// TIA Portal V20 export
FUNCTION_BLOCK "EventsPFE"   // FB74, LAD
AUTHOR : ERsystem_FA2_DH. Kim
// stored: IsIECCheckEnabled true, MemoryReserve 100, Namespace Unit1.Em6, SetENOAutomatically false
   VAR
      data : Array[1..100] of LReal;
   END_VAR
BEGIN

REGION Network 1: Call PFE Events
   // Add the required PFE Events
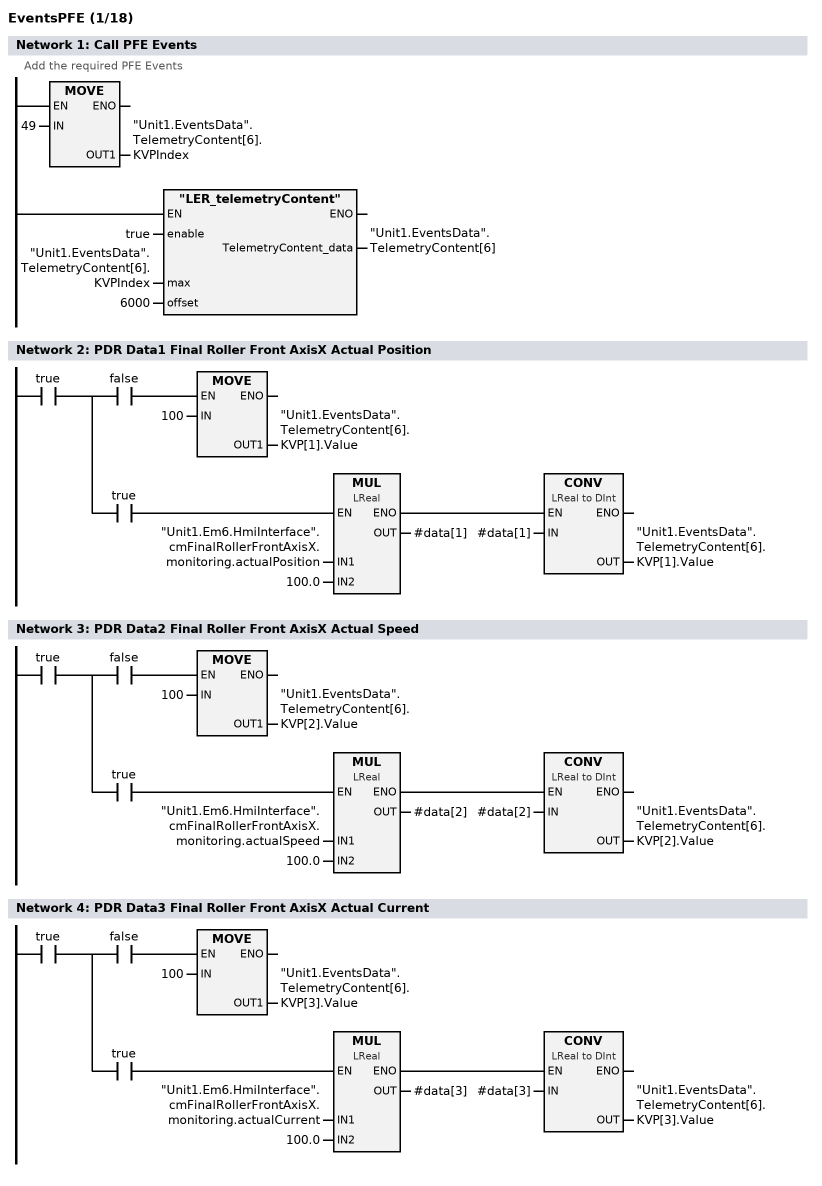
   RUNG wire#powerrail
      Move(in := 49, out1 => "Unit1.EventsData".TelemetryContent[6].KVPIndex)
   END_RUNG
   RUNG wire#powerrail
      "LER_telemetryContent"(enable := true, max := "Unit1.EventsData".TelemetryContent[6].KVPIndex, offset := 6000, TelemetryContent_data => "Unit1.EventsData".TelemetryContent[6])
   END_RUNG
   // the same network as SCL:
   "Unit1.EventsData".TelemetryContent[6].KVPIndex := 49;
   "LER_telemetryContent"(enable := true,
                          max := "Unit1.EventsData".TelemetryContent[6].KVPIndex,
                          offset := 6000,
                          TelemetryContent_data => "Unit1.EventsData".TelemetryContent[6]);
END_REGION

REGION Network 2: PDR Data1 Final Roller Front AxisX Actual Position
   RUNG wire#powerrail
      Contact( true )
      wire#w1
      Contact( false )
      Move(in := 100, out1 => "Unit1.EventsData".TelemetryContent[6].KVP[1].Value)
   END_RUNG
   RUNG wire#w1
      Contact( true )
      { S7_Templates := "SrcType := LReal" } Mul(in1 := "Unit1.Em6.HmiInterface".cmFinalRollerFrontAxisX.monitoring.actualPosition, in2 := 100.0, out => #data[1])
      { S7_Templates := "[SrcType := LReal, DestType := DInt]" } Convert(in := #data[1], out => "Unit1.EventsData".TelemetryContent[6].KVP[1].Value)
   END_RUNG
   // the same network as SCL:
   IF true AND false THEN "Unit1.EventsData".TelemetryContent[6].KVP[1].Value := 100; END_IF;
   IF true AND true THEN
       #data[1] := "Unit1.Em6.HmiInterface".cmFinalRollerFrontAxisX.monitoring.actualPosition * 100.0;
       "Unit1.EventsData".TelemetryContent[6].KVP[1].Value := LREAL_TO_DINT(#data[1]);
   END_IF;
END_REGION

REGION Network 3: PDR Data2 Final Roller Front AxisX Actual Speed
   RUNG wire#powerrail
      Contact( true )
      wire#w1
      Contact( false )
      Move(in := 100, out1 => "Unit1.EventsData".TelemetryContent[6].KVP[2].Value)
   END_RUNG
   RUNG wire#w1
      Contact( true )
      { S7_Templates := "SrcType := LReal" } Mul(in1 := "Unit1.Em6.HmiInterface".cmFinalRollerFrontAxisX.monitoring.actualSpeed, in2 := 100.0, out => #data[2])
      { S7_Templates := "[SrcType := LReal, DestType := DInt]" } Convert(in := #data[2], out => "Unit1.EventsData".TelemetryContent[6].KVP[2].Value)
   END_RUNG
   // the same network as SCL:
   IF true AND false THEN "Unit1.EventsData".TelemetryContent[6].KVP[2].Value := 100; END_IF;
   IF true AND true THEN
       #data[2] := "Unit1.Em6.HmiInterface".cmFinalRollerFrontAxisX.monitoring.actualSpeed * 100.0;
       "Unit1.EventsData".TelemetryContent[6].KVP[2].Value := LREAL_TO_DINT(#data[2]);
   END_IF;
END_REGION

REGION Network 4: PDR Data3 Final Roller Front AxisX Actual Current
   RUNG wire#powerrail
      Contact( true )
      wire#w1
      Contact( false )
      Move(in := 100, out1 => "Unit1.EventsData".TelemetryContent[6].KVP[3].Value)
   END_RUNG
   RUNG wire#w1
      Contact( true )
      { S7_Templates := "SrcType := LReal" } Mul(in1 := "Unit1.Em6.HmiInterface".cmFinalRollerFrontAxisX.monitoring.actualCurrent, in2 := 100.0, out => #data[3])
      { S7_Templates := "[SrcType := LReal, DestType := DInt]" } Convert(in := #data[3], out => "Unit1.EventsData".TelemetryContent[6].KVP[3].Value)
   END_RUNG
   // the same network as SCL:
   IF true AND false THEN "Unit1.EventsData".TelemetryContent[6].KVP[3].Value := 100; END_IF;
   IF true AND true THEN
       #data[3] := "Unit1.Em6.HmiInterface".cmFinalRollerFrontAxisX.monitoring.actualCurrent * 100.0;
       "Unit1.EventsData".TelemetryContent[6].KVP[3].Value := LREAL_TO_DINT(#data[3]);
   END_IF;
END_REGION

REGION Network 5: PDR Data4 Final Roller Front AxisX Actual Torque
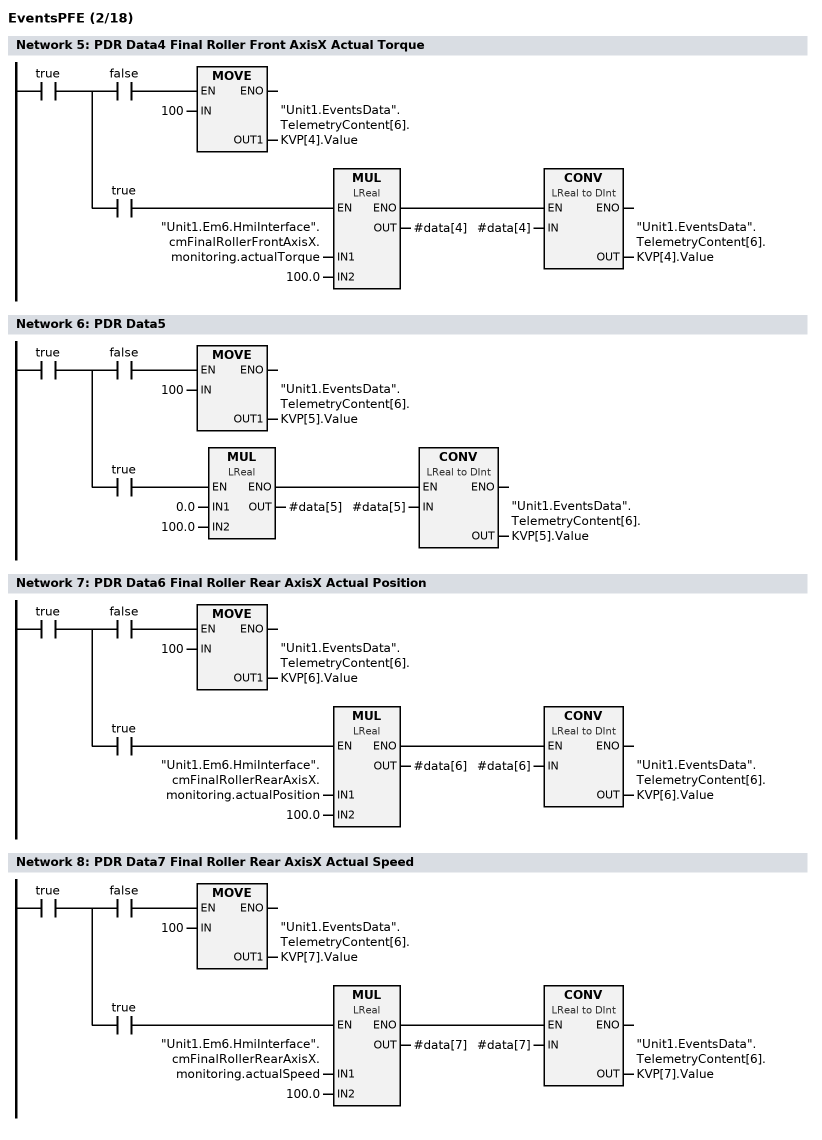
   RUNG wire#powerrail
      Contact( true )
      wire#w1
      Contact( false )
      Move(in := 100, out1 => "Unit1.EventsData".TelemetryContent[6].KVP[4].Value)
   END_RUNG
   RUNG wire#w1
      Contact( true )
      { S7_Templates := "SrcType := LReal" } Mul(in1 := "Unit1.Em6.HmiInterface".cmFinalRollerFrontAxisX.monitoring.actualTorque, in2 := 100.0, out => #data[4])
      { S7_Templates := "[SrcType := LReal, DestType := DInt]" } Convert(in := #data[4], out => "Unit1.EventsData".TelemetryContent[6].KVP[4].Value)
   END_RUNG
   // the same network as SCL:
   IF true AND false THEN "Unit1.EventsData".TelemetryContent[6].KVP[4].Value := 100; END_IF;
   IF true AND true THEN
       #data[4] := "Unit1.Em6.HmiInterface".cmFinalRollerFrontAxisX.monitoring.actualTorque * 100.0;
       "Unit1.EventsData".TelemetryContent[6].KVP[4].Value := LREAL_TO_DINT(#data[4]);
   END_IF;
END_REGION

REGION Network 6: PDR Data5
   RUNG wire#powerrail
      Contact( true )
      wire#w1
      Contact( false )
      Move(in := 100, out1 => "Unit1.EventsData".TelemetryContent[6].KVP[5].Value)
   END_RUNG
   RUNG wire#w1
      Contact( true )
      { S7_Templates := "SrcType := LReal" } Mul(in1 := 0.0, in2 := 100.0, out => #data[5])
      { S7_Templates := "[SrcType := LReal, DestType := DInt]" } Convert(in := #data[5], out => "Unit1.EventsData".TelemetryContent[6].KVP[5].Value)
   END_RUNG
   // the same network as SCL:
   IF true AND false THEN "Unit1.EventsData".TelemetryContent[6].KVP[5].Value := 100; END_IF;
   IF true AND true THEN
       #data[5] := 0.0 * 100.0;
       "Unit1.EventsData".TelemetryContent[6].KVP[5].Value := LREAL_TO_DINT(#data[5]);
   END_IF;
END_REGION

REGION Network 7: PDR Data6 Final Roller Rear AxisX Actual Position
   RUNG wire#powerrail
      Contact( true )
      wire#w1
      Contact( false )
      Move(in := 100, out1 => "Unit1.EventsData".TelemetryContent[6].KVP[6].Value)
   END_RUNG
   RUNG wire#w1
      Contact( true )
      { S7_Templates := "SrcType := LReal" } Mul(in1 := "Unit1.Em6.HmiInterface".cmFinalRollerRearAxisX.monitoring.actualPosition, in2 := 100.0, out => #data[6])
      { S7_Templates := "[SrcType := LReal, DestType := DInt]" } Convert(in := #data[6], out => "Unit1.EventsData".TelemetryContent[6].KVP[6].Value)
   END_RUNG
   // the same network as SCL:
   IF true AND false THEN "Unit1.EventsData".TelemetryContent[6].KVP[6].Value := 100; END_IF;
   IF true AND true THEN
       #data[6] := "Unit1.Em6.HmiInterface".cmFinalRollerRearAxisX.monitoring.actualPosition * 100.0;
       "Unit1.EventsData".TelemetryContent[6].KVP[6].Value := LREAL_TO_DINT(#data[6]);
   END_IF;
END_REGION

REGION Network 8: PDR Data7 Final Roller Rear AxisX Actual Speed
   RUNG wire#powerrail
      Contact( true )
      wire#w1
      Contact( false )
      Move(in := 100, out1 => "Unit1.EventsData".TelemetryContent[6].KVP[7].Value)
   END_RUNG
   RUNG wire#w1
      Contact( true )
      { S7_Templates := "SrcType := LReal" } Mul(in1 := "Unit1.Em6.HmiInterface".cmFinalRollerRearAxisX.monitoring.actualSpeed, in2 := 100.0, out => #data[7])
      { S7_Templates := "[SrcType := LReal, DestType := DInt]" } Convert(in := #data[7], out => "Unit1.EventsData".TelemetryContent[6].KVP[7].Value)
   END_RUNG
   // the same network as SCL:
   IF true AND false THEN "Unit1.EventsData".TelemetryContent[6].KVP[7].Value := 100; END_IF;
   IF true AND true THEN
       #data[7] := "Unit1.Em6.HmiInterface".cmFinalRollerRearAxisX.monitoring.actualSpeed * 100.0;
       "Unit1.EventsData".TelemetryContent[6].KVP[7].Value := LREAL_TO_DINT(#data[7]);
   END_IF;
END_REGION

REGION Network 9: PDR Data8 Final Roller Rear AxisX Actual Current
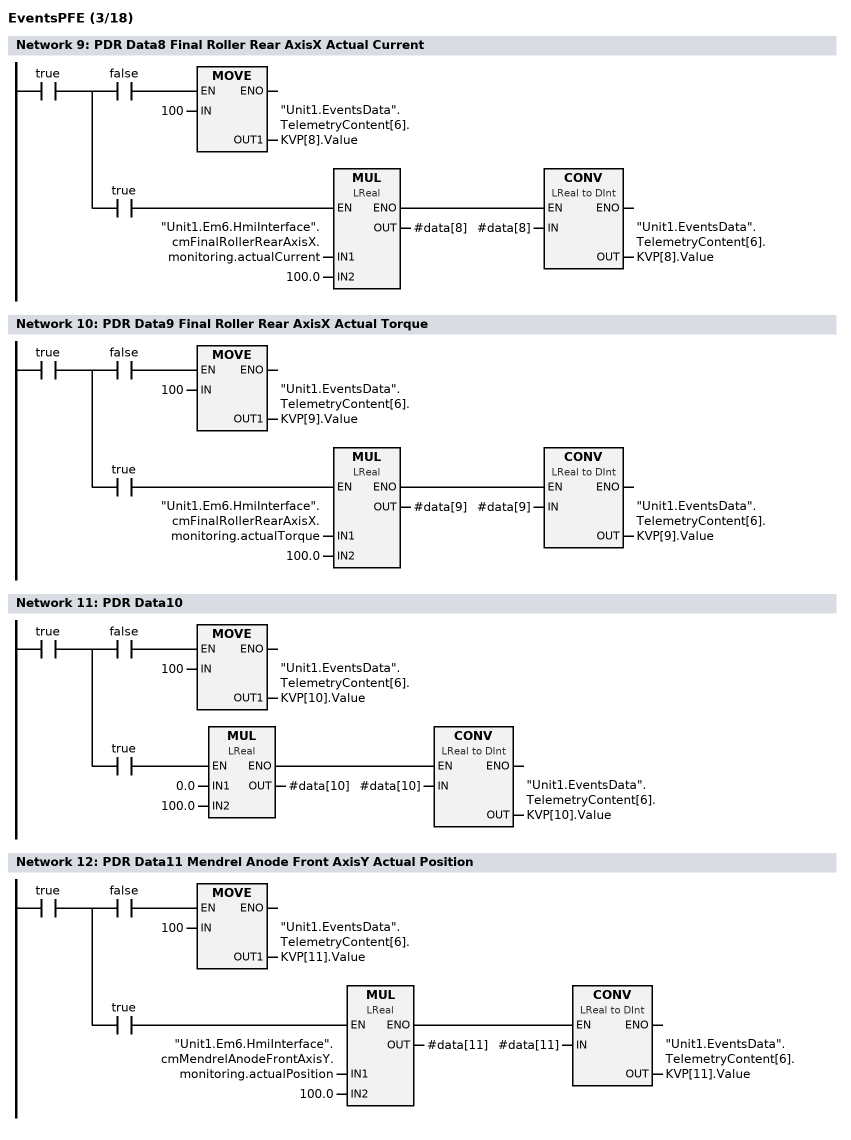
   RUNG wire#powerrail
      Contact( true )
      wire#w1
      Contact( false )
      Move(in := 100, out1 => "Unit1.EventsData".TelemetryContent[6].KVP[8].Value)
   END_RUNG
   RUNG wire#w1
      Contact( true )
      { S7_Templates := "SrcType := LReal" } Mul(in1 := "Unit1.Em6.HmiInterface".cmFinalRollerRearAxisX.monitoring.actualCurrent, in2 := 100.0, out => #data[8])
      { S7_Templates := "[SrcType := LReal, DestType := DInt]" } Convert(in := #data[8], out => "Unit1.EventsData".TelemetryContent[6].KVP[8].Value)
   END_RUNG
   // the same network as SCL:
   IF true AND false THEN "Unit1.EventsData".TelemetryContent[6].KVP[8].Value := 100; END_IF;
   IF true AND true THEN
       #data[8] := "Unit1.Em6.HmiInterface".cmFinalRollerRearAxisX.monitoring.actualCurrent * 100.0;
       "Unit1.EventsData".TelemetryContent[6].KVP[8].Value := LREAL_TO_DINT(#data[8]);
   END_IF;
END_REGION

REGION Network 10: PDR Data9 Final Roller Rear AxisX Actual Torque
   RUNG wire#powerrail
      Contact( true )
      wire#w1
      Contact( false )
      Move(in := 100, out1 => "Unit1.EventsData".TelemetryContent[6].KVP[9].Value)
   END_RUNG
   RUNG wire#w1
      Contact( true )
      { S7_Templates := "SrcType := LReal" } Mul(in1 := "Unit1.Em6.HmiInterface".cmFinalRollerRearAxisX.monitoring.actualTorque, in2 := 100.0, out => #data[9])
      { S7_Templates := "[SrcType := LReal, DestType := DInt]" } Convert(in := #data[9], out => "Unit1.EventsData".TelemetryContent[6].KVP[9].Value)
   END_RUNG
   // the same network as SCL:
   IF true AND false THEN "Unit1.EventsData".TelemetryContent[6].KVP[9].Value := 100; END_IF;
   IF true AND true THEN
       #data[9] := "Unit1.Em6.HmiInterface".cmFinalRollerRearAxisX.monitoring.actualTorque * 100.0;
       "Unit1.EventsData".TelemetryContent[6].KVP[9].Value := LREAL_TO_DINT(#data[9]);
   END_IF;
END_REGION

REGION Network 11: PDR Data10
   RUNG wire#powerrail
      Contact( true )
      wire#w1
      Contact( false )
      Move(in := 100, out1 => "Unit1.EventsData".TelemetryContent[6].KVP[10].Value)
   END_RUNG
   RUNG wire#w1
      Contact( true )
      { S7_Templates := "SrcType := LReal" } Mul(in1 := 0.0, in2 := 100.0, out => #data[10])
      { S7_Templates := "[SrcType := LReal, DestType := DInt]" } Convert(in := #data[10], out => "Unit1.EventsData".TelemetryContent[6].KVP[10].Value)
   END_RUNG
   // the same network as SCL:
   IF true AND false THEN "Unit1.EventsData".TelemetryContent[6].KVP[10].Value := 100; END_IF;
   IF true AND true THEN
       #data[10] := 0.0 * 100.0;
       "Unit1.EventsData".TelemetryContent[6].KVP[10].Value := LREAL_TO_DINT(#data[10]);
   END_IF;
END_REGION

REGION Network 12: PDR Data11 Mendrel Anode Front AxisY Actual Position
   RUNG wire#powerrail
      Contact( true )
      wire#w1
      Contact( false )
      Move(in := 100, out1 => "Unit1.EventsData".TelemetryContent[6].KVP[11].Value)
   END_RUNG
   RUNG wire#w1
      Contact( true )
      { S7_Templates := "SrcType := LReal" } Mul(in1 := "Unit1.Em6.HmiInterface".cmMendrelAnodeFrontAxisY.monitoring.actualPosition, in2 := 100.0, out => #data[11])
      { S7_Templates := "[SrcType := LReal, DestType := DInt]" } Convert(in := #data[11], out => "Unit1.EventsData".TelemetryContent[6].KVP[11].Value)
   END_RUNG
   // the same network as SCL:
   IF true AND false THEN "Unit1.EventsData".TelemetryContent[6].KVP[11].Value := 100; END_IF;
   IF true AND true THEN
       #data[11] := "Unit1.Em6.HmiInterface".cmMendrelAnodeFrontAxisY.monitoring.actualPosition * 100.0;
       "Unit1.EventsData".TelemetryContent[6].KVP[11].Value := LREAL_TO_DINT(#data[11]);
   END_IF;
END_REGION

REGION Network 13: PDR Data12 Mendrel Anode Front AxisY Actual Speed
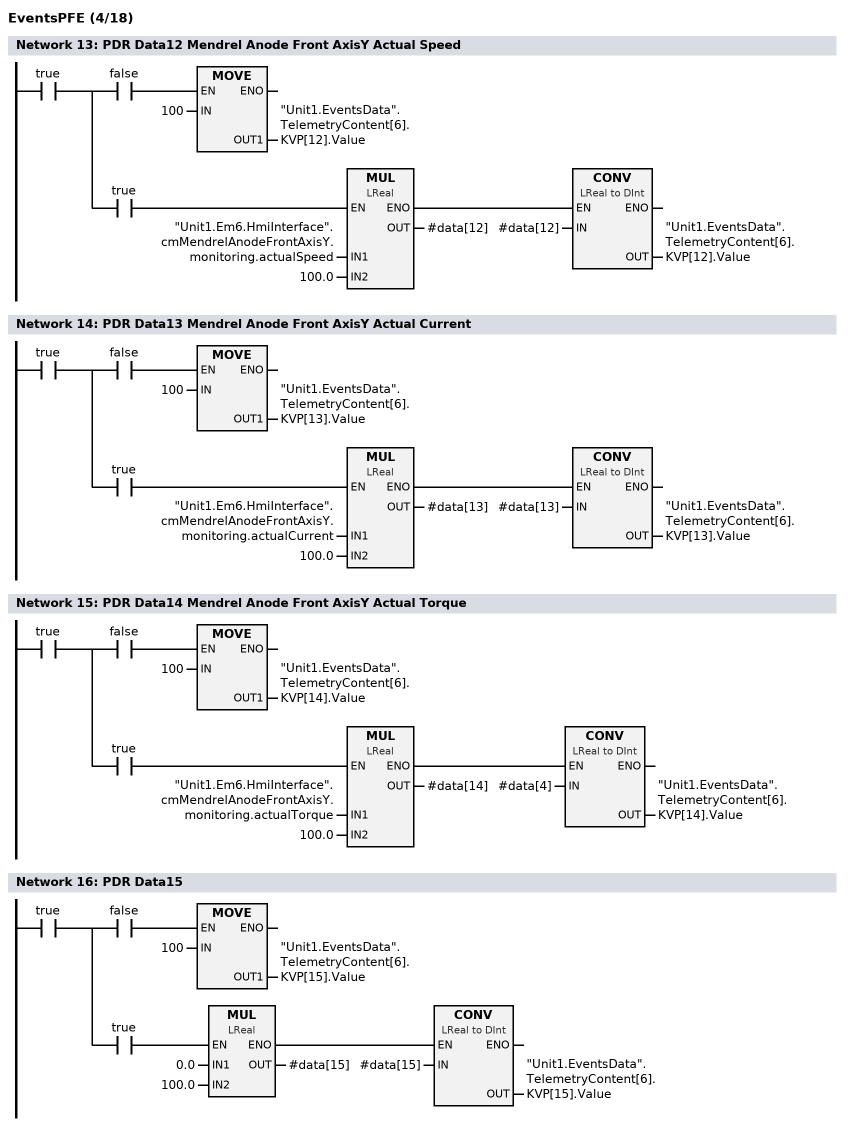
   RUNG wire#powerrail
      Contact( true )
      wire#w1
      Contact( false )
      Move(in := 100, out1 => "Unit1.EventsData".TelemetryContent[6].KVP[12].Value)
   END_RUNG
   RUNG wire#w1
      Contact( true )
      { S7_Templates := "SrcType := LReal" } Mul(in1 := "Unit1.Em6.HmiInterface".cmMendrelAnodeFrontAxisY.monitoring.actualSpeed, in2 := 100.0, out => #data[12])
      { S7_Templates := "[SrcType := LReal, DestType := DInt]" } Convert(in := #data[12], out => "Unit1.EventsData".TelemetryContent[6].KVP[12].Value)
   END_RUNG
   // the same network as SCL:
   IF true AND false THEN "Unit1.EventsData".TelemetryContent[6].KVP[12].Value := 100; END_IF;
   IF true AND true THEN
       #data[12] := "Unit1.Em6.HmiInterface".cmMendrelAnodeFrontAxisY.monitoring.actualSpeed * 100.0;
       "Unit1.EventsData".TelemetryContent[6].KVP[12].Value := LREAL_TO_DINT(#data[12]);
   END_IF;
END_REGION

REGION Network 14: PDR Data13 Mendrel Anode Front AxisY Actual Current
   RUNG wire#powerrail
      Contact( true )
      wire#w1
      Contact( false )
      Move(in := 100, out1 => "Unit1.EventsData".TelemetryContent[6].KVP[13].Value)
   END_RUNG
   RUNG wire#w1
      Contact( true )
      { S7_Templates := "SrcType := LReal" } Mul(in1 := "Unit1.Em6.HmiInterface".cmMendrelAnodeFrontAxisY.monitoring.actualCurrent, in2 := 100.0, out => #data[13])
      { S7_Templates := "[SrcType := LReal, DestType := DInt]" } Convert(in := #data[13], out => "Unit1.EventsData".TelemetryContent[6].KVP[13].Value)
   END_RUNG
   // the same network as SCL:
   IF true AND false THEN "Unit1.EventsData".TelemetryContent[6].KVP[13].Value := 100; END_IF;
   IF true AND true THEN
       #data[13] := "Unit1.Em6.HmiInterface".cmMendrelAnodeFrontAxisY.monitoring.actualCurrent * 100.0;
       "Unit1.EventsData".TelemetryContent[6].KVP[13].Value := LREAL_TO_DINT(#data[13]);
   END_IF;
END_REGION

REGION Network 15: PDR Data14 Mendrel Anode Front AxisY Actual Torque
   RUNG wire#powerrail
      Contact( true )
      wire#w1
      Contact( false )
      Move(in := 100, out1 => "Unit1.EventsData".TelemetryContent[6].KVP[14].Value)
   END_RUNG
   RUNG wire#w1
      Contact( true )
      { S7_Templates := "SrcType := LReal" } Mul(in1 := "Unit1.Em6.HmiInterface".cmMendrelAnodeFrontAxisY.monitoring.actualTorque, in2 := 100.0, out => #data[14])
      { S7_Templates := "[SrcType := LReal, DestType := DInt]" } Convert(in := #data[4], out => "Unit1.EventsData".TelemetryContent[6].KVP[14].Value)
   END_RUNG
   // the same network as SCL:
   IF true AND false THEN "Unit1.EventsData".TelemetryContent[6].KVP[14].Value := 100; END_IF;
   IF true AND true THEN
       #data[14] := "Unit1.Em6.HmiInterface".cmMendrelAnodeFrontAxisY.monitoring.actualTorque * 100.0;
       "Unit1.EventsData".TelemetryContent[6].KVP[14].Value := LREAL_TO_DINT(#data[4]);
   END_IF;
END_REGION

REGION Network 16: PDR Data15
   RUNG wire#powerrail
      Contact( true )
      wire#w1
      Contact( false )
      Move(in := 100, out1 => "Unit1.EventsData".TelemetryContent[6].KVP[15].Value)
   END_RUNG
   RUNG wire#w1
      Contact( true )
      { S7_Templates := "SrcType := LReal" } Mul(in1 := 0.0, in2 := 100.0, out => #data[15])
      { S7_Templates := "[SrcType := LReal, DestType := DInt]" } Convert(in := #data[15], out => "Unit1.EventsData".TelemetryContent[6].KVP[15].Value)
   END_RUNG
   // the same network as SCL:
   IF true AND false THEN "Unit1.EventsData".TelemetryContent[6].KVP[15].Value := 100; END_IF;
   IF true AND true THEN
       #data[15] := 0.0 * 100.0;
       "Unit1.EventsData".TelemetryContent[6].KVP[15].Value := LREAL_TO_DINT(#data[15]);
   END_IF;
END_REGION

REGION Network 17: PDR Data16 Mendrel Anode Front AxisZ Actual Position
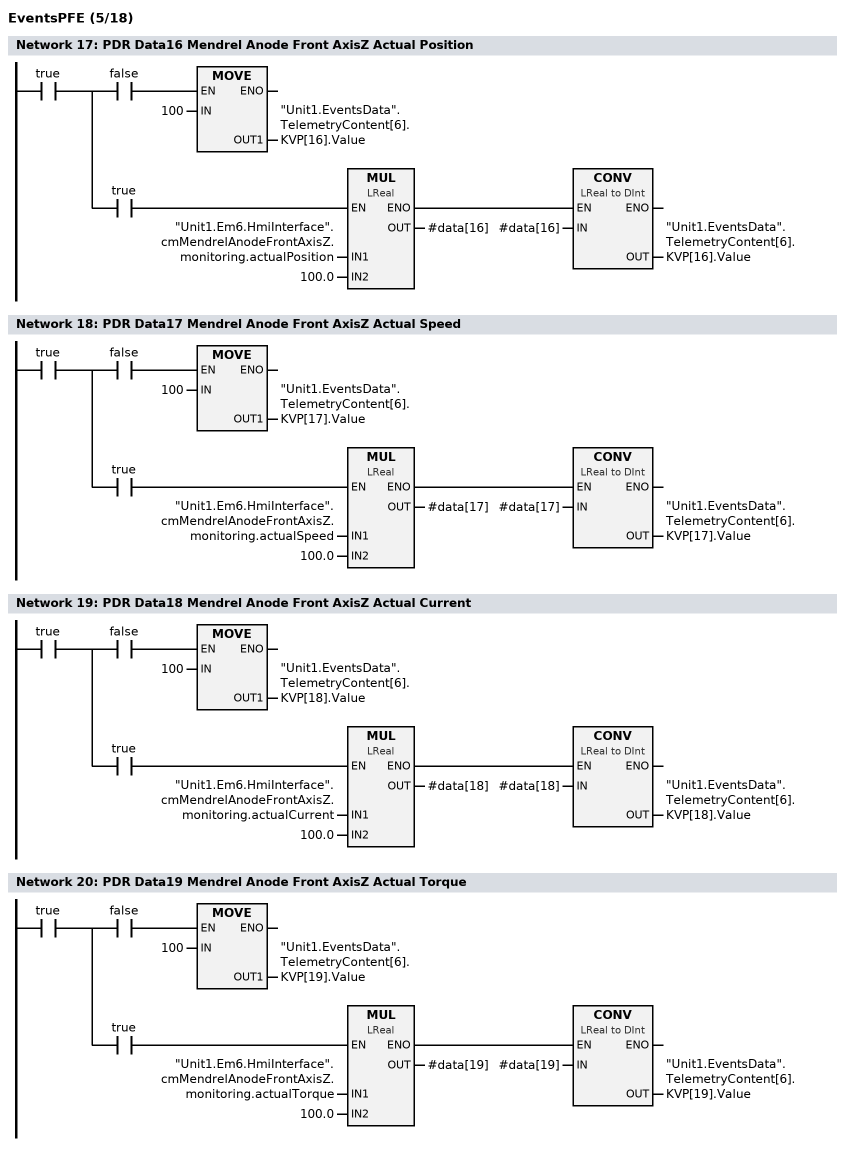
   RUNG wire#powerrail
      Contact( true )
      wire#w1
      Contact( false )
      Move(in := 100, out1 => "Unit1.EventsData".TelemetryContent[6].KVP[16].Value)
   END_RUNG
   RUNG wire#w1
      Contact( true )
      { S7_Templates := "SrcType := LReal" } Mul(in1 := "Unit1.Em6.HmiInterface".cmMendrelAnodeFrontAxisZ.monitoring.actualPosition, in2 := 100.0, out => #data[16])
      { S7_Templates := "[SrcType := LReal, DestType := DInt]" } Convert(in := #data[16], out => "Unit1.EventsData".TelemetryContent[6].KVP[16].Value)
   END_RUNG
   // the same network as SCL:
   IF true AND false THEN "Unit1.EventsData".TelemetryContent[6].KVP[16].Value := 100; END_IF;
   IF true AND true THEN
       #data[16] := "Unit1.Em6.HmiInterface".cmMendrelAnodeFrontAxisZ.monitoring.actualPosition * 100.0;
       "Unit1.EventsData".TelemetryContent[6].KVP[16].Value := LREAL_TO_DINT(#data[16]);
   END_IF;
END_REGION

REGION Network 18: PDR Data17 Mendrel Anode Front AxisZ Actual Speed
   RUNG wire#powerrail
      Contact( true )
      wire#w1
      Contact( false )
      Move(in := 100, out1 => "Unit1.EventsData".TelemetryContent[6].KVP[17].Value)
   END_RUNG
   RUNG wire#w1
      Contact( true )
      { S7_Templates := "SrcType := LReal" } Mul(in1 := "Unit1.Em6.HmiInterface".cmMendrelAnodeFrontAxisZ.monitoring.actualSpeed, in2 := 100.0, out => #data[17])
      { S7_Templates := "[SrcType := LReal, DestType := DInt]" } Convert(in := #data[17], out => "Unit1.EventsData".TelemetryContent[6].KVP[17].Value)
   END_RUNG
   // the same network as SCL:
   IF true AND false THEN "Unit1.EventsData".TelemetryContent[6].KVP[17].Value := 100; END_IF;
   IF true AND true THEN
       #data[17] := "Unit1.Em6.HmiInterface".cmMendrelAnodeFrontAxisZ.monitoring.actualSpeed * 100.0;
       "Unit1.EventsData".TelemetryContent[6].KVP[17].Value := LREAL_TO_DINT(#data[17]);
   END_IF;
END_REGION

REGION Network 19: PDR Data18 Mendrel Anode Front AxisZ Actual Current
   RUNG wire#powerrail
      Contact( true )
      wire#w1
      Contact( false )
      Move(in := 100, out1 => "Unit1.EventsData".TelemetryContent[6].KVP[18].Value)
   END_RUNG
   RUNG wire#w1
      Contact( true )
      { S7_Templates := "SrcType := LReal" } Mul(in1 := "Unit1.Em6.HmiInterface".cmMendrelAnodeFrontAxisZ.monitoring.actualCurrent, in2 := 100.0, out => #data[18])
      { S7_Templates := "[SrcType := LReal, DestType := DInt]" } Convert(in := #data[18], out => "Unit1.EventsData".TelemetryContent[6].KVP[18].Value)
   END_RUNG
   // the same network as SCL:
   IF true AND false THEN "Unit1.EventsData".TelemetryContent[6].KVP[18].Value := 100; END_IF;
   IF true AND true THEN
       #data[18] := "Unit1.Em6.HmiInterface".cmMendrelAnodeFrontAxisZ.monitoring.actualCurrent * 100.0;
       "Unit1.EventsData".TelemetryContent[6].KVP[18].Value := LREAL_TO_DINT(#data[18]);
   END_IF;
END_REGION

REGION Network 20: PDR Data19 Mendrel Anode Front AxisZ Actual Torque
   RUNG wire#powerrail
      Contact( true )
      wire#w1
      Contact( false )
      Move(in := 100, out1 => "Unit1.EventsData".TelemetryContent[6].KVP[19].Value)
   END_RUNG
   RUNG wire#w1
      Contact( true )
      { S7_Templates := "SrcType := LReal" } Mul(in1 := "Unit1.Em6.HmiInterface".cmMendrelAnodeFrontAxisZ.monitoring.actualTorque, in2 := 100.0, out => #data[19])
      { S7_Templates := "[SrcType := LReal, DestType := DInt]" } Convert(in := #data[19], out => "Unit1.EventsData".TelemetryContent[6].KVP[19].Value)
   END_RUNG
   // the same network as SCL:
   IF true AND false THEN "Unit1.EventsData".TelemetryContent[6].KVP[19].Value := 100; END_IF;
   IF true AND true THEN
       #data[19] := "Unit1.Em6.HmiInterface".cmMendrelAnodeFrontAxisZ.monitoring.actualTorque * 100.0;
       "Unit1.EventsData".TelemetryContent[6].KVP[19].Value := LREAL_TO_DINT(#data[19]);
   END_IF;
END_REGION

REGION Network 21: PDR Data20
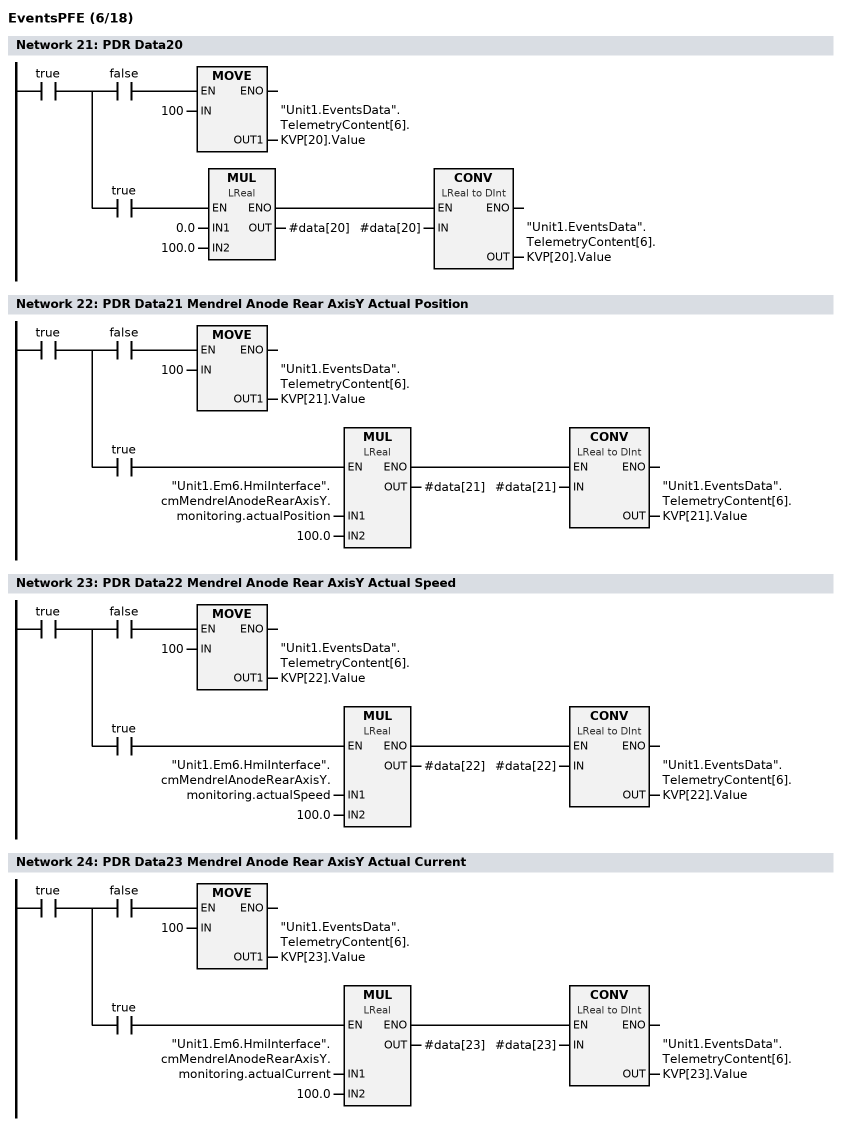
   RUNG wire#powerrail
      Contact( true )
      wire#w1
      Contact( false )
      Move(in := 100, out1 => "Unit1.EventsData".TelemetryContent[6].KVP[20].Value)
   END_RUNG
   RUNG wire#w1
      Contact( true )
      { S7_Templates := "SrcType := LReal" } Mul(in1 := 0.0, in2 := 100.0, out => #data[20])
      { S7_Templates := "[SrcType := LReal, DestType := DInt]" } Convert(in := #data[20], out => "Unit1.EventsData".TelemetryContent[6].KVP[20].Value)
   END_RUNG
   // the same network as SCL:
   IF true AND false THEN "Unit1.EventsData".TelemetryContent[6].KVP[20].Value := 100; END_IF;
   IF true AND true THEN
       #data[20] := 0.0 * 100.0;
       "Unit1.EventsData".TelemetryContent[6].KVP[20].Value := LREAL_TO_DINT(#data[20]);
   END_IF;
END_REGION

REGION Network 22: PDR Data21 Mendrel Anode Rear AxisY Actual Position
   RUNG wire#powerrail
      Contact( true )
      wire#w1
      Contact( false )
      Move(in := 100, out1 => "Unit1.EventsData".TelemetryContent[6].KVP[21].Value)
   END_RUNG
   RUNG wire#w1
      Contact( true )
      { S7_Templates := "SrcType := LReal" } Mul(in1 := "Unit1.Em6.HmiInterface".cmMendrelAnodeRearAxisY.monitoring.actualPosition, in2 := 100.0, out => #data[21])
      { S7_Templates := "[SrcType := LReal, DestType := DInt]" } Convert(in := #data[21], out => "Unit1.EventsData".TelemetryContent[6].KVP[21].Value)
   END_RUNG
   // the same network as SCL:
   IF true AND false THEN "Unit1.EventsData".TelemetryContent[6].KVP[21].Value := 100; END_IF;
   IF true AND true THEN
       #data[21] := "Unit1.Em6.HmiInterface".cmMendrelAnodeRearAxisY.monitoring.actualPosition * 100.0;
       "Unit1.EventsData".TelemetryContent[6].KVP[21].Value := LREAL_TO_DINT(#data[21]);
   END_IF;
END_REGION

REGION Network 23: PDR Data22 Mendrel Anode Rear AxisY Actual Speed
   RUNG wire#powerrail
      Contact( true )
      wire#w1
      Contact( false )
      Move(in := 100, out1 => "Unit1.EventsData".TelemetryContent[6].KVP[22].Value)
   END_RUNG
   RUNG wire#w1
      Contact( true )
      { S7_Templates := "SrcType := LReal" } Mul(in1 := "Unit1.Em6.HmiInterface".cmMendrelAnodeRearAxisY.monitoring.actualSpeed, in2 := 100.0, out => #data[22])
      { S7_Templates := "[SrcType := LReal, DestType := DInt]" } Convert(in := #data[22], out => "Unit1.EventsData".TelemetryContent[6].KVP[22].Value)
   END_RUNG
   // the same network as SCL:
   IF true AND false THEN "Unit1.EventsData".TelemetryContent[6].KVP[22].Value := 100; END_IF;
   IF true AND true THEN
       #data[22] := "Unit1.Em6.HmiInterface".cmMendrelAnodeRearAxisY.monitoring.actualSpeed * 100.0;
       "Unit1.EventsData".TelemetryContent[6].KVP[22].Value := LREAL_TO_DINT(#data[22]);
   END_IF;
END_REGION

REGION Network 24: PDR Data23 Mendrel Anode Rear AxisY Actual Current
   RUNG wire#powerrail
      Contact( true )
      wire#w1
      Contact( false )
      Move(in := 100, out1 => "Unit1.EventsData".TelemetryContent[6].KVP[23].Value)
   END_RUNG
   RUNG wire#w1
      Contact( true )
      { S7_Templates := "SrcType := LReal" } Mul(in1 := "Unit1.Em6.HmiInterface".cmMendrelAnodeRearAxisY.monitoring.actualCurrent, in2 := 100.0, out => #data[23])
      { S7_Templates := "[SrcType := LReal, DestType := DInt]" } Convert(in := #data[23], out => "Unit1.EventsData".TelemetryContent[6].KVP[23].Value)
   END_RUNG
   // the same network as SCL:
   IF true AND false THEN "Unit1.EventsData".TelemetryContent[6].KVP[23].Value := 100; END_IF;
   IF true AND true THEN
       #data[23] := "Unit1.Em6.HmiInterface".cmMendrelAnodeRearAxisY.monitoring.actualCurrent * 100.0;
       "Unit1.EventsData".TelemetryContent[6].KVP[23].Value := LREAL_TO_DINT(#data[23]);
   END_IF;
END_REGION

REGION Network 25: PDR Data24 Mendrel Anode Rear AxisY Actual Torque
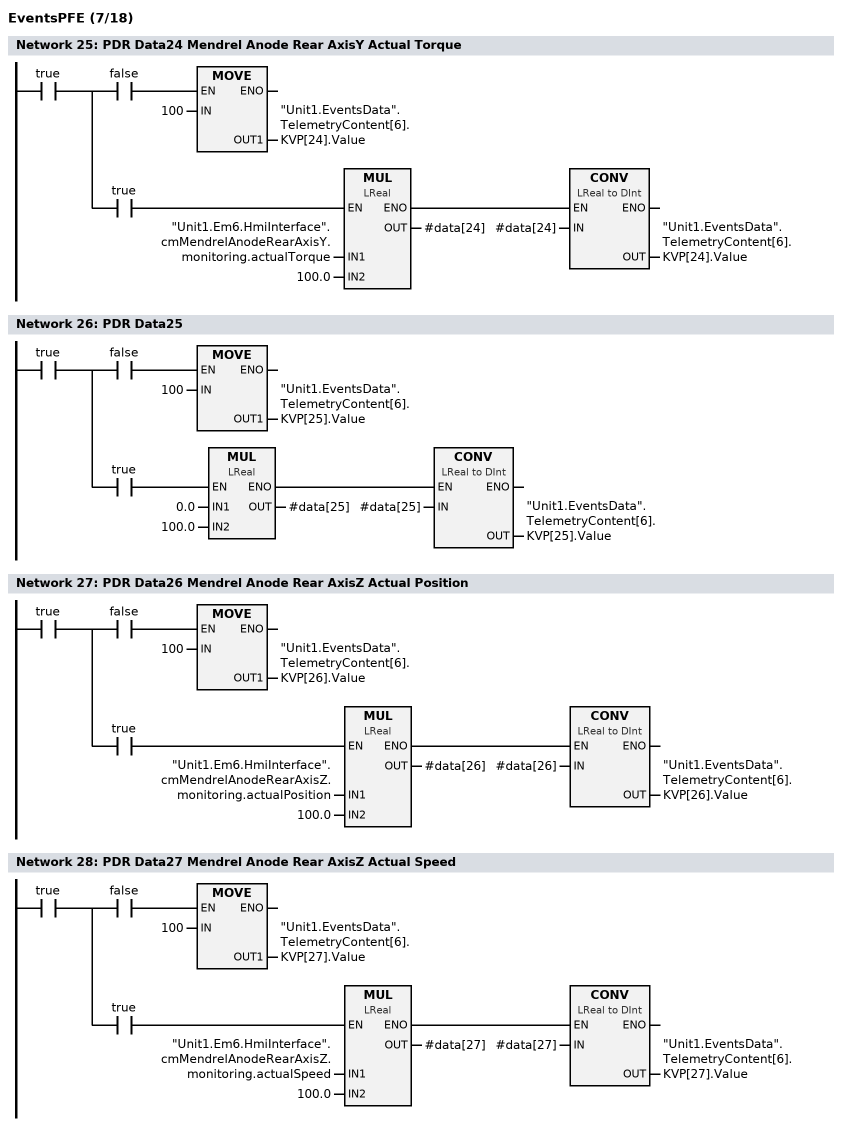
   RUNG wire#powerrail
      Contact( true )
      wire#w1
      Contact( false )
      Move(in := 100, out1 => "Unit1.EventsData".TelemetryContent[6].KVP[24].Value)
   END_RUNG
   RUNG wire#w1
      Contact( true )
      { S7_Templates := "SrcType := LReal" } Mul(in1 := "Unit1.Em6.HmiInterface".cmMendrelAnodeRearAxisY.monitoring.actualTorque, in2 := 100.0, out => #data[24])
      { S7_Templates := "[SrcType := LReal, DestType := DInt]" } Convert(in := #data[24], out => "Unit1.EventsData".TelemetryContent[6].KVP[24].Value)
   END_RUNG
   // the same network as SCL:
   IF true AND false THEN "Unit1.EventsData".TelemetryContent[6].KVP[24].Value := 100; END_IF;
   IF true AND true THEN
       #data[24] := "Unit1.Em6.HmiInterface".cmMendrelAnodeRearAxisY.monitoring.actualTorque * 100.0;
       "Unit1.EventsData".TelemetryContent[6].KVP[24].Value := LREAL_TO_DINT(#data[24]);
   END_IF;
END_REGION

REGION Network 26: PDR Data25
   RUNG wire#powerrail
      Contact( true )
      wire#w1
      Contact( false )
      Move(in := 100, out1 => "Unit1.EventsData".TelemetryContent[6].KVP[25].Value)
   END_RUNG
   RUNG wire#w1
      Contact( true )
      { S7_Templates := "SrcType := LReal" } Mul(in1 := 0.0, in2 := 100.0, out => #data[25])
      { S7_Templates := "[SrcType := LReal, DestType := DInt]" } Convert(in := #data[25], out => "Unit1.EventsData".TelemetryContent[6].KVP[25].Value)
   END_RUNG
   // the same network as SCL:
   IF true AND false THEN "Unit1.EventsData".TelemetryContent[6].KVP[25].Value := 100; END_IF;
   IF true AND true THEN
       #data[25] := 0.0 * 100.0;
       "Unit1.EventsData".TelemetryContent[6].KVP[25].Value := LREAL_TO_DINT(#data[25]);
   END_IF;
END_REGION

REGION Network 27: PDR Data26 Mendrel Anode Rear AxisZ Actual Position
   RUNG wire#powerrail
      Contact( true )
      wire#w1
      Contact( false )
      Move(in := 100, out1 => "Unit1.EventsData".TelemetryContent[6].KVP[26].Value)
   END_RUNG
   RUNG wire#w1
      Contact( true )
      { S7_Templates := "SrcType := LReal" } Mul(in1 := "Unit1.Em6.HmiInterface".cmMendrelAnodeRearAxisZ.monitoring.actualPosition, in2 := 100.0, out => #data[26])
      { S7_Templates := "[SrcType := LReal, DestType := DInt]" } Convert(in := #data[26], out => "Unit1.EventsData".TelemetryContent[6].KVP[26].Value)
   END_RUNG
   // the same network as SCL:
   IF true AND false THEN "Unit1.EventsData".TelemetryContent[6].KVP[26].Value := 100; END_IF;
   IF true AND true THEN
       #data[26] := "Unit1.Em6.HmiInterface".cmMendrelAnodeRearAxisZ.monitoring.actualPosition * 100.0;
       "Unit1.EventsData".TelemetryContent[6].KVP[26].Value := LREAL_TO_DINT(#data[26]);
   END_IF;
END_REGION

REGION Network 28: PDR Data27 Mendrel Anode Rear AxisZ Actual Speed
   RUNG wire#powerrail
      Contact( true )
      wire#w1
      Contact( false )
      Move(in := 100, out1 => "Unit1.EventsData".TelemetryContent[6].KVP[27].Value)
   END_RUNG
   RUNG wire#w1
      Contact( true )
      { S7_Templates := "SrcType := LReal" } Mul(in1 := "Unit1.Em6.HmiInterface".cmMendrelAnodeRearAxisZ.monitoring.actualSpeed, in2 := 100.0, out => #data[27])
      { S7_Templates := "[SrcType := LReal, DestType := DInt]" } Convert(in := #data[27], out => "Unit1.EventsData".TelemetryContent[6].KVP[27].Value)
   END_RUNG
   // the same network as SCL:
   IF true AND false THEN "Unit1.EventsData".TelemetryContent[6].KVP[27].Value := 100; END_IF;
   IF true AND true THEN
       #data[27] := "Unit1.Em6.HmiInterface".cmMendrelAnodeRearAxisZ.monitoring.actualSpeed * 100.0;
       "Unit1.EventsData".TelemetryContent[6].KVP[27].Value := LREAL_TO_DINT(#data[27]);
   END_IF;
END_REGION

REGION Network 29: PDR Data28 Mendrel Anode Rear AxisZ Actual Current
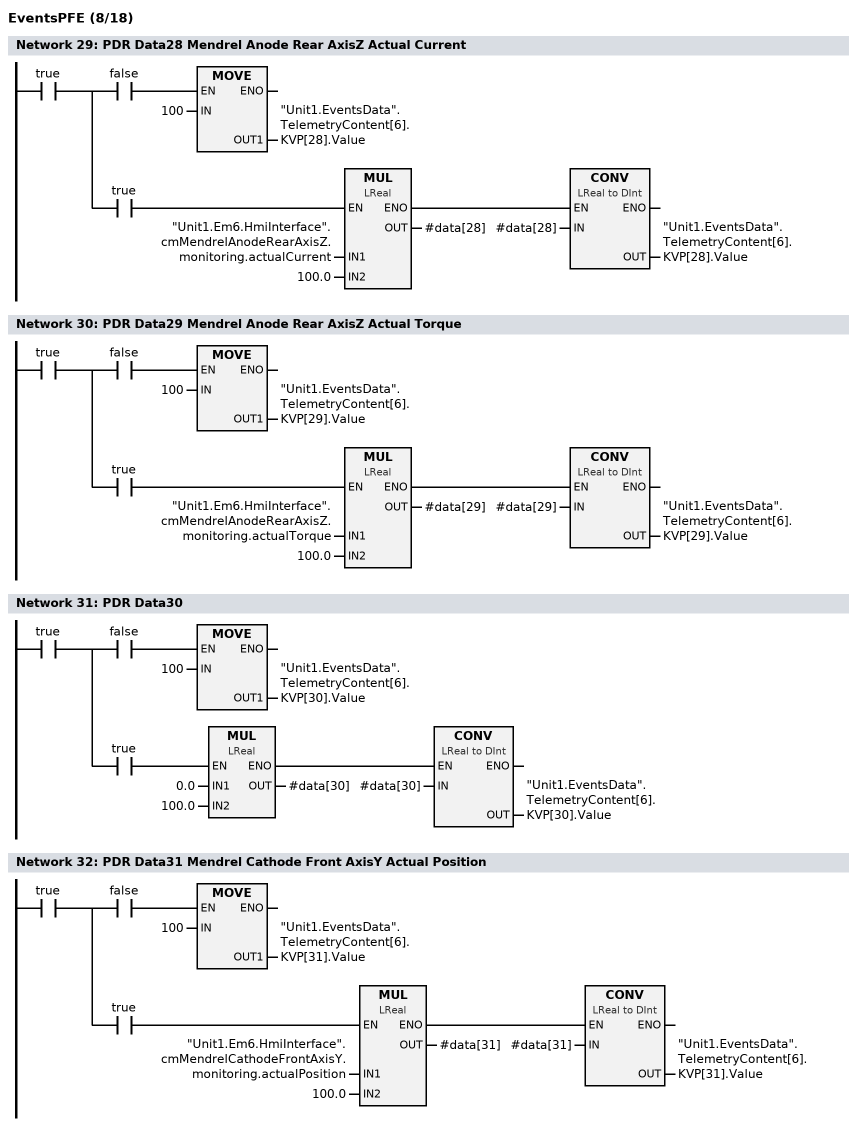
   RUNG wire#powerrail
      Contact( true )
      wire#w1
      Contact( false )
      Move(in := 100, out1 => "Unit1.EventsData".TelemetryContent[6].KVP[28].Value)
   END_RUNG
   RUNG wire#w1
      Contact( true )
      { S7_Templates := "SrcType := LReal" } Mul(in1 := "Unit1.Em6.HmiInterface".cmMendrelAnodeRearAxisZ.monitoring.actualCurrent, in2 := 100.0, out => #data[28])
      { S7_Templates := "[SrcType := LReal, DestType := DInt]" } Convert(in := #data[28], out => "Unit1.EventsData".TelemetryContent[6].KVP[28].Value)
   END_RUNG
   // the same network as SCL:
   IF true AND false THEN "Unit1.EventsData".TelemetryContent[6].KVP[28].Value := 100; END_IF;
   IF true AND true THEN
       #data[28] := "Unit1.Em6.HmiInterface".cmMendrelAnodeRearAxisZ.monitoring.actualCurrent * 100.0;
       "Unit1.EventsData".TelemetryContent[6].KVP[28].Value := LREAL_TO_DINT(#data[28]);
   END_IF;
END_REGION

REGION Network 30: PDR Data29 Mendrel Anode Rear AxisZ Actual Torque
   RUNG wire#powerrail
      Contact( true )
      wire#w1
      Contact( false )
      Move(in := 100, out1 => "Unit1.EventsData".TelemetryContent[6].KVP[29].Value)
   END_RUNG
   RUNG wire#w1
      Contact( true )
      { S7_Templates := "SrcType := LReal" } Mul(in1 := "Unit1.Em6.HmiInterface".cmMendrelAnodeRearAxisZ.monitoring.actualTorque, in2 := 100.0, out => #data[29])
      { S7_Templates := "[SrcType := LReal, DestType := DInt]" } Convert(in := #data[29], out => "Unit1.EventsData".TelemetryContent[6].KVP[29].Value)
   END_RUNG
   // the same network as SCL:
   IF true AND false THEN "Unit1.EventsData".TelemetryContent[6].KVP[29].Value := 100; END_IF;
   IF true AND true THEN
       #data[29] := "Unit1.Em6.HmiInterface".cmMendrelAnodeRearAxisZ.monitoring.actualTorque * 100.0;
       "Unit1.EventsData".TelemetryContent[6].KVP[29].Value := LREAL_TO_DINT(#data[29]);
   END_IF;
END_REGION

REGION Network 31: PDR Data30
   RUNG wire#powerrail
      Contact( true )
      wire#w1
      Contact( false )
      Move(in := 100, out1 => "Unit1.EventsData".TelemetryContent[6].KVP[30].Value)
   END_RUNG
   RUNG wire#w1
      Contact( true )
      { S7_Templates := "SrcType := LReal" } Mul(in1 := 0.0, in2 := 100.0, out => #data[30])
      { S7_Templates := "[SrcType := LReal, DestType := DInt]" } Convert(in := #data[30], out => "Unit1.EventsData".TelemetryContent[6].KVP[30].Value)
   END_RUNG
   // the same network as SCL:
   IF true AND false THEN "Unit1.EventsData".TelemetryContent[6].KVP[30].Value := 100; END_IF;
   IF true AND true THEN
       #data[30] := 0.0 * 100.0;
       "Unit1.EventsData".TelemetryContent[6].KVP[30].Value := LREAL_TO_DINT(#data[30]);
   END_IF;
END_REGION

REGION Network 32: PDR Data31 Mendrel Cathode Front AxisY Actual Position
   RUNG wire#powerrail
      Contact( true )
      wire#w1
      Contact( false )
      Move(in := 100, out1 => "Unit1.EventsData".TelemetryContent[6].KVP[31].Value)
   END_RUNG
   RUNG wire#w1
      Contact( true )
      { S7_Templates := "SrcType := LReal" } Mul(in1 := "Unit1.Em6.HmiInterface".cmMendrelCathodeFrontAxisY.monitoring.actualPosition, in2 := 100.0, out => #data[31])
      { S7_Templates := "[SrcType := LReal, DestType := DInt]" } Convert(in := #data[31], out => "Unit1.EventsData".TelemetryContent[6].KVP[31].Value)
   END_RUNG
   // the same network as SCL:
   IF true AND false THEN "Unit1.EventsData".TelemetryContent[6].KVP[31].Value := 100; END_IF;
   IF true AND true THEN
       #data[31] := "Unit1.Em6.HmiInterface".cmMendrelCathodeFrontAxisY.monitoring.actualPosition * 100.0;
       "Unit1.EventsData".TelemetryContent[6].KVP[31].Value := LREAL_TO_DINT(#data[31]);
   END_IF;
END_REGION

REGION Network 33: PDR Data32 Mendrel Cathode Front AxisY Actual Speed
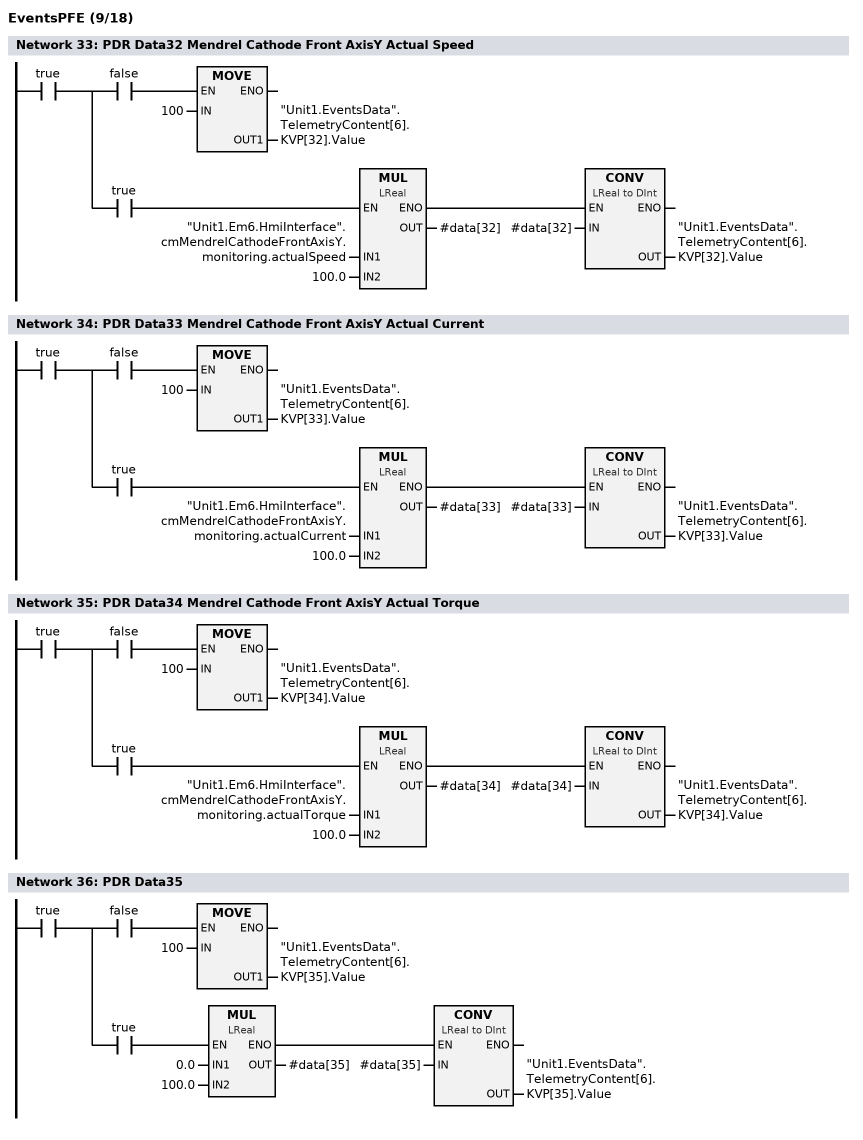
   RUNG wire#powerrail
      Contact( true )
      wire#w1
      Contact( false )
      Move(in := 100, out1 => "Unit1.EventsData".TelemetryContent[6].KVP[32].Value)
   END_RUNG
   RUNG wire#w1
      Contact( true )
      { S7_Templates := "SrcType := LReal" } Mul(in1 := "Unit1.Em6.HmiInterface".cmMendrelCathodeFrontAxisY.monitoring.actualSpeed, in2 := 100.0, out => #data[32])
      { S7_Templates := "[SrcType := LReal, DestType := DInt]" } Convert(in := #data[32], out => "Unit1.EventsData".TelemetryContent[6].KVP[32].Value)
   END_RUNG
   // the same network as SCL:
   IF true AND false THEN "Unit1.EventsData".TelemetryContent[6].KVP[32].Value := 100; END_IF;
   IF true AND true THEN
       #data[32] := "Unit1.Em6.HmiInterface".cmMendrelCathodeFrontAxisY.monitoring.actualSpeed * 100.0;
       "Unit1.EventsData".TelemetryContent[6].KVP[32].Value := LREAL_TO_DINT(#data[32]);
   END_IF;
END_REGION

REGION Network 34: PDR Data33 Mendrel Cathode Front AxisY Actual Current
   RUNG wire#powerrail
      Contact( true )
      wire#w1
      Contact( false )
      Move(in := 100, out1 => "Unit1.EventsData".TelemetryContent[6].KVP[33].Value)
   END_RUNG
   RUNG wire#w1
      Contact( true )
      { S7_Templates := "SrcType := LReal" } Mul(in1 := "Unit1.Em6.HmiInterface".cmMendrelCathodeFrontAxisY.monitoring.actualCurrent, in2 := 100.0, out => #data[33])
      { S7_Templates := "[SrcType := LReal, DestType := DInt]" } Convert(in := #data[33], out => "Unit1.EventsData".TelemetryContent[6].KVP[33].Value)
   END_RUNG
   // the same network as SCL:
   IF true AND false THEN "Unit1.EventsData".TelemetryContent[6].KVP[33].Value := 100; END_IF;
   IF true AND true THEN
       #data[33] := "Unit1.Em6.HmiInterface".cmMendrelCathodeFrontAxisY.monitoring.actualCurrent * 100.0;
       "Unit1.EventsData".TelemetryContent[6].KVP[33].Value := LREAL_TO_DINT(#data[33]);
   END_IF;
END_REGION

REGION Network 35: PDR Data34 Mendrel Cathode Front AxisY Actual Torque
   RUNG wire#powerrail
      Contact( true )
      wire#w1
      Contact( false )
      Move(in := 100, out1 => "Unit1.EventsData".TelemetryContent[6].KVP[34].Value)
   END_RUNG
   RUNG wire#w1
      Contact( true )
      { S7_Templates := "SrcType := LReal" } Mul(in1 := "Unit1.Em6.HmiInterface".cmMendrelCathodeFrontAxisY.monitoring.actualTorque, in2 := 100.0, out => #data[34])
      { S7_Templates := "[SrcType := LReal, DestType := DInt]" } Convert(in := #data[34], out => "Unit1.EventsData".TelemetryContent[6].KVP[34].Value)
   END_RUNG
   // the same network as SCL:
   IF true AND false THEN "Unit1.EventsData".TelemetryContent[6].KVP[34].Value := 100; END_IF;
   IF true AND true THEN
       #data[34] := "Unit1.Em6.HmiInterface".cmMendrelCathodeFrontAxisY.monitoring.actualTorque * 100.0;
       "Unit1.EventsData".TelemetryContent[6].KVP[34].Value := LREAL_TO_DINT(#data[34]);
   END_IF;
END_REGION

REGION Network 36: PDR Data35
   RUNG wire#powerrail
      Contact( true )
      wire#w1
      Contact( false )
      Move(in := 100, out1 => "Unit1.EventsData".TelemetryContent[6].KVP[35].Value)
   END_RUNG
   RUNG wire#w1
      Contact( true )
      { S7_Templates := "SrcType := LReal" } Mul(in1 := 0.0, in2 := 100.0, out => #data[35])
      { S7_Templates := "[SrcType := LReal, DestType := DInt]" } Convert(in := #data[35], out => "Unit1.EventsData".TelemetryContent[6].KVP[35].Value)
   END_RUNG
   // the same network as SCL:
   IF true AND false THEN "Unit1.EventsData".TelemetryContent[6].KVP[35].Value := 100; END_IF;
   IF true AND true THEN
       #data[35] := 0.0 * 100.0;
       "Unit1.EventsData".TelemetryContent[6].KVP[35].Value := LREAL_TO_DINT(#data[35]);
   END_IF;
END_REGION

REGION Network 37: PDR Data36 Mendrel Cathode Front AxisZ Actual Position
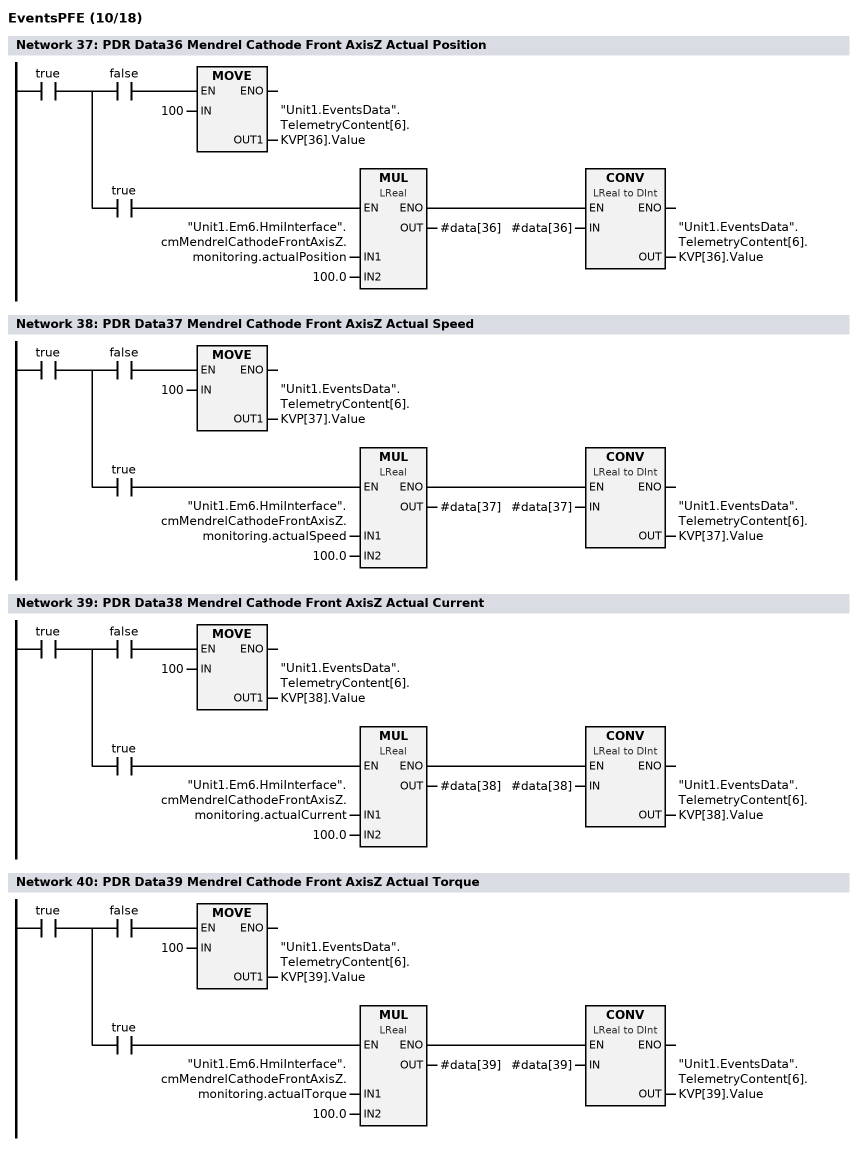
   RUNG wire#powerrail
      Contact( true )
      wire#w1
      Contact( false )
      Move(in := 100, out1 => "Unit1.EventsData".TelemetryContent[6].KVP[36].Value)
   END_RUNG
   RUNG wire#w1
      Contact( true )
      { S7_Templates := "SrcType := LReal" } Mul(in1 := "Unit1.Em6.HmiInterface".cmMendrelCathodeFrontAxisZ.monitoring.actualPosition, in2 := 100.0, out => #data[36])
      { S7_Templates := "[SrcType := LReal, DestType := DInt]" } Convert(in := #data[36], out => "Unit1.EventsData".TelemetryContent[6].KVP[36].Value)
   END_RUNG
   // the same network as SCL:
   IF true AND false THEN "Unit1.EventsData".TelemetryContent[6].KVP[36].Value := 100; END_IF;
   IF true AND true THEN
       #data[36] := "Unit1.Em6.HmiInterface".cmMendrelCathodeFrontAxisZ.monitoring.actualPosition * 100.0;
       "Unit1.EventsData".TelemetryContent[6].KVP[36].Value := LREAL_TO_DINT(#data[36]);
   END_IF;
END_REGION

REGION Network 38: PDR Data37 Mendrel Cathode Front AxisZ Actual Speed
   RUNG wire#powerrail
      Contact( true )
      wire#w1
      Contact( false )
      Move(in := 100, out1 => "Unit1.EventsData".TelemetryContent[6].KVP[37].Value)
   END_RUNG
   RUNG wire#w1
      Contact( true )
      { S7_Templates := "SrcType := LReal" } Mul(in1 := "Unit1.Em6.HmiInterface".cmMendrelCathodeFrontAxisZ.monitoring.actualSpeed, in2 := 100.0, out => #data[37])
      { S7_Templates := "[SrcType := LReal, DestType := DInt]" } Convert(in := #data[37], out => "Unit1.EventsData".TelemetryContent[6].KVP[37].Value)
   END_RUNG
   // the same network as SCL:
   IF true AND false THEN "Unit1.EventsData".TelemetryContent[6].KVP[37].Value := 100; END_IF;
   IF true AND true THEN
       #data[37] := "Unit1.Em6.HmiInterface".cmMendrelCathodeFrontAxisZ.monitoring.actualSpeed * 100.0;
       "Unit1.EventsData".TelemetryContent[6].KVP[37].Value := LREAL_TO_DINT(#data[37]);
   END_IF;
END_REGION

REGION Network 39: PDR Data38 Mendrel Cathode Front AxisZ Actual Current
   RUNG wire#powerrail
      Contact( true )
      wire#w1
      Contact( false )
      Move(in := 100, out1 => "Unit1.EventsData".TelemetryContent[6].KVP[38].Value)
   END_RUNG
   RUNG wire#w1
      Contact( true )
      { S7_Templates := "SrcType := LReal" } Mul(in1 := "Unit1.Em6.HmiInterface".cmMendrelCathodeFrontAxisZ.monitoring.actualCurrent, in2 := 100.0, out => #data[38])
      { S7_Templates := "[SrcType := LReal, DestType := DInt]" } Convert(in := #data[38], out => "Unit1.EventsData".TelemetryContent[6].KVP[38].Value)
   END_RUNG
   // the same network as SCL:
   IF true AND false THEN "Unit1.EventsData".TelemetryContent[6].KVP[38].Value := 100; END_IF;
   IF true AND true THEN
       #data[38] := "Unit1.Em6.HmiInterface".cmMendrelCathodeFrontAxisZ.monitoring.actualCurrent * 100.0;
       "Unit1.EventsData".TelemetryContent[6].KVP[38].Value := LREAL_TO_DINT(#data[38]);
   END_IF;
END_REGION

REGION Network 40: PDR Data39 Mendrel Cathode Front AxisZ Actual Torque
   RUNG wire#powerrail
      Contact( true )
      wire#w1
      Contact( false )
      Move(in := 100, out1 => "Unit1.EventsData".TelemetryContent[6].KVP[39].Value)
   END_RUNG
   RUNG wire#w1
      Contact( true )
      { S7_Templates := "SrcType := LReal" } Mul(in1 := "Unit1.Em6.HmiInterface".cmMendrelCathodeFrontAxisZ.monitoring.actualTorque, in2 := 100.0, out => #data[39])
      { S7_Templates := "[SrcType := LReal, DestType := DInt]" } Convert(in := #data[39], out => "Unit1.EventsData".TelemetryContent[6].KVP[39].Value)
   END_RUNG
   // the same network as SCL:
   IF true AND false THEN "Unit1.EventsData".TelemetryContent[6].KVP[39].Value := 100; END_IF;
   IF true AND true THEN
       #data[39] := "Unit1.Em6.HmiInterface".cmMendrelCathodeFrontAxisZ.monitoring.actualTorque * 100.0;
       "Unit1.EventsData".TelemetryContent[6].KVP[39].Value := LREAL_TO_DINT(#data[39]);
   END_IF;
END_REGION

REGION Network 41: PDR Data40
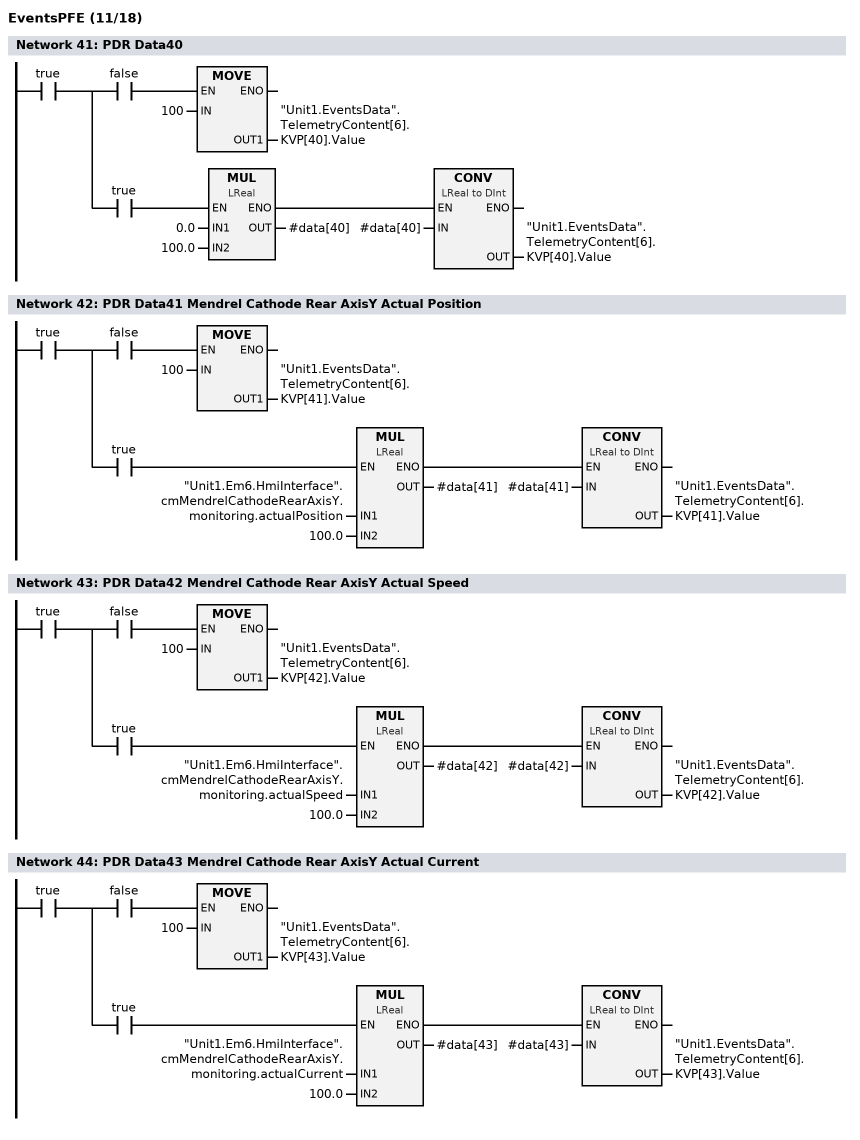
   RUNG wire#powerrail
      Contact( true )
      wire#w1
      Contact( false )
      Move(in := 100, out1 => "Unit1.EventsData".TelemetryContent[6].KVP[40].Value)
   END_RUNG
   RUNG wire#w1
      Contact( true )
      { S7_Templates := "SrcType := LReal" } Mul(in1 := 0.0, in2 := 100.0, out => #data[40])
      { S7_Templates := "[SrcType := LReal, DestType := DInt]" } Convert(in := #data[40], out => "Unit1.EventsData".TelemetryContent[6].KVP[40].Value)
   END_RUNG
   // the same network as SCL:
   IF true AND false THEN "Unit1.EventsData".TelemetryContent[6].KVP[40].Value := 100; END_IF;
   IF true AND true THEN
       #data[40] := 0.0 * 100.0;
       "Unit1.EventsData".TelemetryContent[6].KVP[40].Value := LREAL_TO_DINT(#data[40]);
   END_IF;
END_REGION

REGION Network 42: PDR Data41 Mendrel Cathode Rear AxisY Actual Position
   RUNG wire#powerrail
      Contact( true )
      wire#w1
      Contact( false )
      Move(in := 100, out1 => "Unit1.EventsData".TelemetryContent[6].KVP[41].Value)
   END_RUNG
   RUNG wire#w1
      Contact( true )
      { S7_Templates := "SrcType := LReal" } Mul(in1 := "Unit1.Em6.HmiInterface".cmMendrelCathodeRearAxisY.monitoring.actualPosition, in2 := 100.0, out => #data[41])
      { S7_Templates := "[SrcType := LReal, DestType := DInt]" } Convert(in := #data[41], out => "Unit1.EventsData".TelemetryContent[6].KVP[41].Value)
   END_RUNG
   // the same network as SCL:
   IF true AND false THEN "Unit1.EventsData".TelemetryContent[6].KVP[41].Value := 100; END_IF;
   IF true AND true THEN
       #data[41] := "Unit1.Em6.HmiInterface".cmMendrelCathodeRearAxisY.monitoring.actualPosition * 100.0;
       "Unit1.EventsData".TelemetryContent[6].KVP[41].Value := LREAL_TO_DINT(#data[41]);
   END_IF;
END_REGION

REGION Network 43: PDR Data42 Mendrel Cathode Rear AxisY Actual Speed
   RUNG wire#powerrail
      Contact( true )
      wire#w1
      Contact( false )
      Move(in := 100, out1 => "Unit1.EventsData".TelemetryContent[6].KVP[42].Value)
   END_RUNG
   RUNG wire#w1
      Contact( true )
      { S7_Templates := "SrcType := LReal" } Mul(in1 := "Unit1.Em6.HmiInterface".cmMendrelCathodeRearAxisY.monitoring.actualSpeed, in2 := 100.0, out => #data[42])
      { S7_Templates := "[SrcType := LReal, DestType := DInt]" } Convert(in := #data[42], out => "Unit1.EventsData".TelemetryContent[6].KVP[42].Value)
   END_RUNG
   // the same network as SCL:
   IF true AND false THEN "Unit1.EventsData".TelemetryContent[6].KVP[42].Value := 100; END_IF;
   IF true AND true THEN
       #data[42] := "Unit1.Em6.HmiInterface".cmMendrelCathodeRearAxisY.monitoring.actualSpeed * 100.0;
       "Unit1.EventsData".TelemetryContent[6].KVP[42].Value := LREAL_TO_DINT(#data[42]);
   END_IF;
END_REGION

REGION Network 44: PDR Data43 Mendrel Cathode Rear AxisY Actual Current
   RUNG wire#powerrail
      Contact( true )
      wire#w1
      Contact( false )
      Move(in := 100, out1 => "Unit1.EventsData".TelemetryContent[6].KVP[43].Value)
   END_RUNG
   RUNG wire#w1
      Contact( true )
      { S7_Templates := "SrcType := LReal" } Mul(in1 := "Unit1.Em6.HmiInterface".cmMendrelCathodeRearAxisY.monitoring.actualCurrent, in2 := 100.0, out => #data[43])
      { S7_Templates := "[SrcType := LReal, DestType := DInt]" } Convert(in := #data[43], out => "Unit1.EventsData".TelemetryContent[6].KVP[43].Value)
   END_RUNG
   // the same network as SCL:
   IF true AND false THEN "Unit1.EventsData".TelemetryContent[6].KVP[43].Value := 100; END_IF;
   IF true AND true THEN
       #data[43] := "Unit1.Em6.HmiInterface".cmMendrelCathodeRearAxisY.monitoring.actualCurrent * 100.0;
       "Unit1.EventsData".TelemetryContent[6].KVP[43].Value := LREAL_TO_DINT(#data[43]);
   END_IF;
END_REGION

REGION Network 45: PDR Data44 Mendrel Cathode Rear AxisY Actual Torque
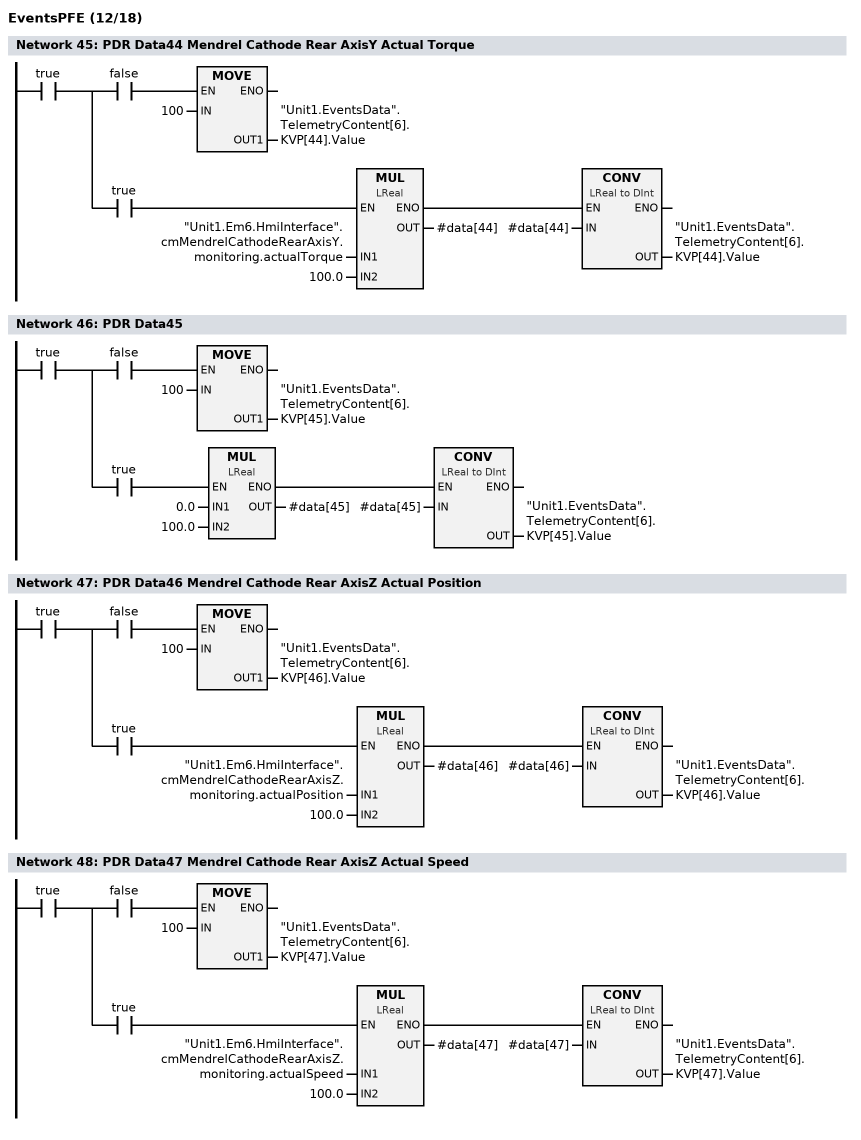
   RUNG wire#powerrail
      Contact( true )
      wire#w1
      Contact( false )
      Move(in := 100, out1 => "Unit1.EventsData".TelemetryContent[6].KVP[44].Value)
   END_RUNG
   RUNG wire#w1
      Contact( true )
      { S7_Templates := "SrcType := LReal" } Mul(in1 := "Unit1.Em6.HmiInterface".cmMendrelCathodeRearAxisY.monitoring.actualTorque, in2 := 100.0, out => #data[44])
      { S7_Templates := "[SrcType := LReal, DestType := DInt]" } Convert(in := #data[44], out => "Unit1.EventsData".TelemetryContent[6].KVP[44].Value)
   END_RUNG
   // the same network as SCL:
   IF true AND false THEN "Unit1.EventsData".TelemetryContent[6].KVP[44].Value := 100; END_IF;
   IF true AND true THEN
       #data[44] := "Unit1.Em6.HmiInterface".cmMendrelCathodeRearAxisY.monitoring.actualTorque * 100.0;
       "Unit1.EventsData".TelemetryContent[6].KVP[44].Value := LREAL_TO_DINT(#data[44]);
   END_IF;
END_REGION

REGION Network 46: PDR Data45
   RUNG wire#powerrail
      Contact( true )
      wire#w1
      Contact( false )
      Move(in := 100, out1 => "Unit1.EventsData".TelemetryContent[6].KVP[45].Value)
   END_RUNG
   RUNG wire#w1
      Contact( true )
      { S7_Templates := "SrcType := LReal" } Mul(in1 := 0.0, in2 := 100.0, out => #data[45])
      { S7_Templates := "[SrcType := LReal, DestType := DInt]" } Convert(in := #data[45], out => "Unit1.EventsData".TelemetryContent[6].KVP[45].Value)
   END_RUNG
   // the same network as SCL:
   IF true AND false THEN "Unit1.EventsData".TelemetryContent[6].KVP[45].Value := 100; END_IF;
   IF true AND true THEN
       #data[45] := 0.0 * 100.0;
       "Unit1.EventsData".TelemetryContent[6].KVP[45].Value := LREAL_TO_DINT(#data[45]);
   END_IF;
END_REGION

REGION Network 47: PDR Data46 Mendrel Cathode Rear AxisZ Actual Position
   RUNG wire#powerrail
      Contact( true )
      wire#w1
      Contact( false )
      Move(in := 100, out1 => "Unit1.EventsData".TelemetryContent[6].KVP[46].Value)
   END_RUNG
   RUNG wire#w1
      Contact( true )
      { S7_Templates := "SrcType := LReal" } Mul(in1 := "Unit1.Em6.HmiInterface".cmMendrelCathodeRearAxisZ.monitoring.actualPosition, in2 := 100.0, out => #data[46])
      { S7_Templates := "[SrcType := LReal, DestType := DInt]" } Convert(in := #data[46], out => "Unit1.EventsData".TelemetryContent[6].KVP[46].Value)
   END_RUNG
   // the same network as SCL:
   IF true AND false THEN "Unit1.EventsData".TelemetryContent[6].KVP[46].Value := 100; END_IF;
   IF true AND true THEN
       #data[46] := "Unit1.Em6.HmiInterface".cmMendrelCathodeRearAxisZ.monitoring.actualPosition * 100.0;
       "Unit1.EventsData".TelemetryContent[6].KVP[46].Value := LREAL_TO_DINT(#data[46]);
   END_IF;
END_REGION

REGION Network 48: PDR Data47 Mendrel Cathode Rear AxisZ Actual Speed
   RUNG wire#powerrail
      Contact( true )
      wire#w1
      Contact( false )
      Move(in := 100, out1 => "Unit1.EventsData".TelemetryContent[6].KVP[47].Value)
   END_RUNG
   RUNG wire#w1
      Contact( true )
      { S7_Templates := "SrcType := LReal" } Mul(in1 := "Unit1.Em6.HmiInterface".cmMendrelCathodeRearAxisZ.monitoring.actualSpeed, in2 := 100.0, out => #data[47])
      { S7_Templates := "[SrcType := LReal, DestType := DInt]" } Convert(in := #data[47], out => "Unit1.EventsData".TelemetryContent[6].KVP[47].Value)
   END_RUNG
   // the same network as SCL:
   IF true AND false THEN "Unit1.EventsData".TelemetryContent[6].KVP[47].Value := 100; END_IF;
   IF true AND true THEN
       #data[47] := "Unit1.Em6.HmiInterface".cmMendrelCathodeRearAxisZ.monitoring.actualSpeed * 100.0;
       "Unit1.EventsData".TelemetryContent[6].KVP[47].Value := LREAL_TO_DINT(#data[47]);
   END_IF;
END_REGION

REGION Network 49: PDR Data48 Mendrel Cathode Rear AxisZ Actual Current
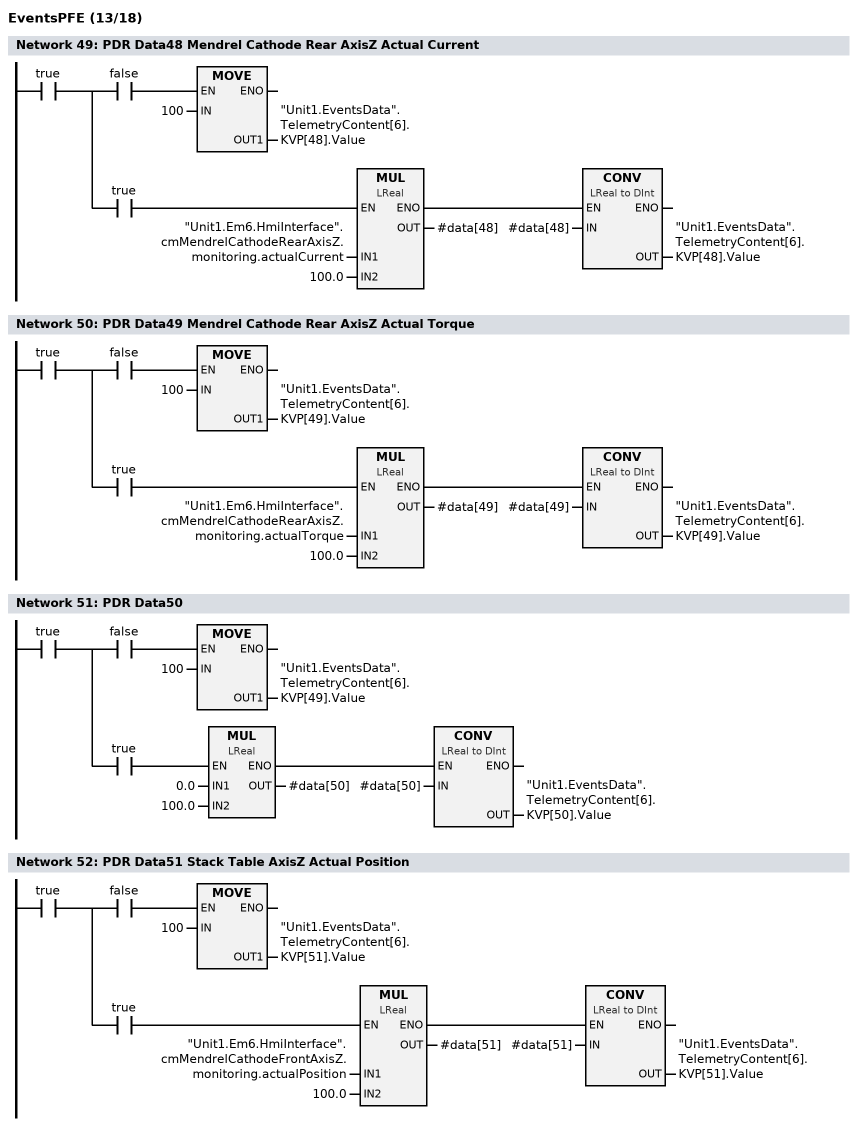
   RUNG wire#powerrail
      Contact( true )
      wire#w1
      Contact( false )
      Move(in := 100, out1 => "Unit1.EventsData".TelemetryContent[6].KVP[48].Value)
   END_RUNG
   RUNG wire#w1
      Contact( true )
      { S7_Templates := "SrcType := LReal" } Mul(in1 := "Unit1.Em6.HmiInterface".cmMendrelCathodeRearAxisZ.monitoring.actualCurrent, in2 := 100.0, out => #data[48])
      { S7_Templates := "[SrcType := LReal, DestType := DInt]" } Convert(in := #data[48], out => "Unit1.EventsData".TelemetryContent[6].KVP[48].Value)
   END_RUNG
   // the same network as SCL:
   IF true AND false THEN "Unit1.EventsData".TelemetryContent[6].KVP[48].Value := 100; END_IF;
   IF true AND true THEN
       #data[48] := "Unit1.Em6.HmiInterface".cmMendrelCathodeRearAxisZ.monitoring.actualCurrent * 100.0;
       "Unit1.EventsData".TelemetryContent[6].KVP[48].Value := LREAL_TO_DINT(#data[48]);
   END_IF;
END_REGION

REGION Network 50: PDR Data49 Mendrel Cathode Rear AxisZ Actual Torque
   RUNG wire#powerrail
      Contact( true )
      wire#w1
      Contact( false )
      Move(in := 100, out1 => "Unit1.EventsData".TelemetryContent[6].KVP[49].Value)
   END_RUNG
   RUNG wire#w1
      Contact( true )
      { S7_Templates := "SrcType := LReal" } Mul(in1 := "Unit1.Em6.HmiInterface".cmMendrelCathodeRearAxisZ.monitoring.actualTorque, in2 := 100.0, out => #data[49])
      { S7_Templates := "[SrcType := LReal, DestType := DInt]" } Convert(in := #data[49], out => "Unit1.EventsData".TelemetryContent[6].KVP[49].Value)
   END_RUNG
   // the same network as SCL:
   IF true AND false THEN "Unit1.EventsData".TelemetryContent[6].KVP[49].Value := 100; END_IF;
   IF true AND true THEN
       #data[49] := "Unit1.Em6.HmiInterface".cmMendrelCathodeRearAxisZ.monitoring.actualTorque * 100.0;
       "Unit1.EventsData".TelemetryContent[6].KVP[49].Value := LREAL_TO_DINT(#data[49]);
   END_IF;
END_REGION

REGION Network 51: PDR Data50
   RUNG wire#powerrail
      Contact( true )
      wire#w1
      Contact( false )
      Move(in := 100, out1 => "Unit1.EventsData".TelemetryContent[6].KVP[49].Value)
   END_RUNG
   RUNG wire#w1
      Contact( true )
      { S7_Templates := "SrcType := LReal" } Mul(in1 := 0.0, in2 := 100.0, out => #data[50])
      { S7_Templates := "[SrcType := LReal, DestType := DInt]" } Convert(in := #data[50], out => "Unit1.EventsData".TelemetryContent[6].KVP[50].Value)
   END_RUNG
   // the same network as SCL:
   IF true AND false THEN "Unit1.EventsData".TelemetryContent[6].KVP[49].Value := 100; END_IF;
   IF true AND true THEN
       #data[50] := 0.0 * 100.0;
       "Unit1.EventsData".TelemetryContent[6].KVP[50].Value := LREAL_TO_DINT(#data[50]);
   END_IF;
END_REGION

REGION Network 52: PDR Data51 Stack Table AxisZ Actual Position
   RUNG wire#powerrail
      Contact( true )
      wire#w1
      Contact( false )
      Move(in := 100, out1 => "Unit1.EventsData".TelemetryContent[6].KVP[51].Value)
   END_RUNG
   RUNG wire#w1
      Contact( true )
      { S7_Templates := "SrcType := LReal" } Mul(in1 := "Unit1.Em6.HmiInterface".cmMendrelCathodeFrontAxisZ.monitoring.actualPosition, in2 := 100.0, out => #data[51])
      { S7_Templates := "[SrcType := LReal, DestType := DInt]" } Convert(in := #data[51], out => "Unit1.EventsData".TelemetryContent[6].KVP[51].Value)
   END_RUNG
   // the same network as SCL:
   IF true AND false THEN "Unit1.EventsData".TelemetryContent[6].KVP[51].Value := 100; END_IF;
   IF true AND true THEN
       #data[51] := "Unit1.Em6.HmiInterface".cmMendrelCathodeFrontAxisZ.monitoring.actualPosition * 100.0;
       "Unit1.EventsData".TelemetryContent[6].KVP[51].Value := LREAL_TO_DINT(#data[51]);
   END_IF;
END_REGION

REGION Network 53: PDR Data52 Stack Table AxisZ Actual Speed
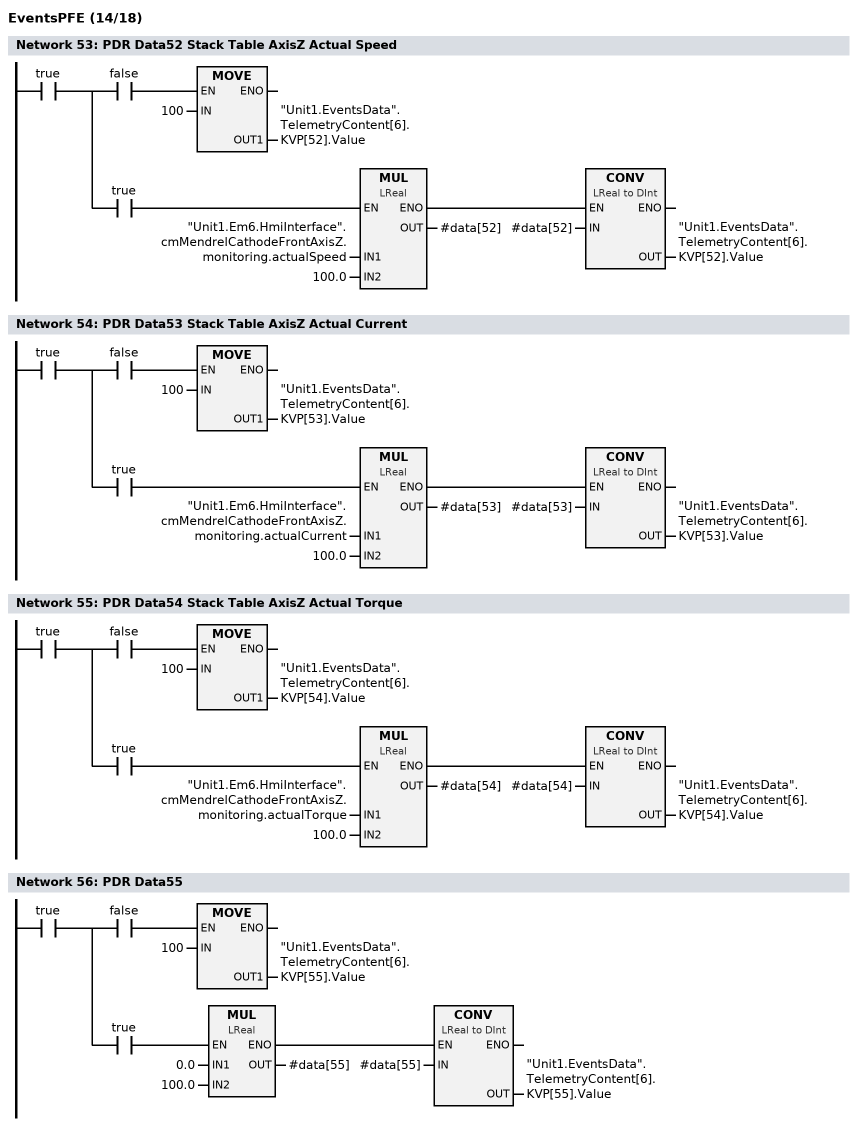
   RUNG wire#powerrail
      Contact( true )
      wire#w1
      Contact( false )
      Move(in := 100, out1 => "Unit1.EventsData".TelemetryContent[6].KVP[52].Value)
   END_RUNG
   RUNG wire#w1
      Contact( true )
      { S7_Templates := "SrcType := LReal" } Mul(in1 := "Unit1.Em6.HmiInterface".cmMendrelCathodeFrontAxisZ.monitoring.actualSpeed, in2 := 100.0, out => #data[52])
      { S7_Templates := "[SrcType := LReal, DestType := DInt]" } Convert(in := #data[52], out => "Unit1.EventsData".TelemetryContent[6].KVP[52].Value)
   END_RUNG
   // the same network as SCL:
   IF true AND false THEN "Unit1.EventsData".TelemetryContent[6].KVP[52].Value := 100; END_IF;
   IF true AND true THEN
       #data[52] := "Unit1.Em6.HmiInterface".cmMendrelCathodeFrontAxisZ.monitoring.actualSpeed * 100.0;
       "Unit1.EventsData".TelemetryContent[6].KVP[52].Value := LREAL_TO_DINT(#data[52]);
   END_IF;
END_REGION

REGION Network 54: PDR Data53 Stack Table AxisZ Actual Current
   RUNG wire#powerrail
      Contact( true )
      wire#w1
      Contact( false )
      Move(in := 100, out1 => "Unit1.EventsData".TelemetryContent[6].KVP[53].Value)
   END_RUNG
   RUNG wire#w1
      Contact( true )
      { S7_Templates := "SrcType := LReal" } Mul(in1 := "Unit1.Em6.HmiInterface".cmMendrelCathodeFrontAxisZ.monitoring.actualCurrent, in2 := 100.0, out => #data[53])
      { S7_Templates := "[SrcType := LReal, DestType := DInt]" } Convert(in := #data[53], out => "Unit1.EventsData".TelemetryContent[6].KVP[53].Value)
   END_RUNG
   // the same network as SCL:
   IF true AND false THEN "Unit1.EventsData".TelemetryContent[6].KVP[53].Value := 100; END_IF;
   IF true AND true THEN
       #data[53] := "Unit1.Em6.HmiInterface".cmMendrelCathodeFrontAxisZ.monitoring.actualCurrent * 100.0;
       "Unit1.EventsData".TelemetryContent[6].KVP[53].Value := LREAL_TO_DINT(#data[53]);
   END_IF;
END_REGION

REGION Network 55: PDR Data54 Stack Table AxisZ Actual Torque
   RUNG wire#powerrail
      Contact( true )
      wire#w1
      Contact( false )
      Move(in := 100, out1 => "Unit1.EventsData".TelemetryContent[6].KVP[54].Value)
   END_RUNG
   RUNG wire#w1
      Contact( true )
      { S7_Templates := "SrcType := LReal" } Mul(in1 := "Unit1.Em6.HmiInterface".cmMendrelCathodeFrontAxisZ.monitoring.actualTorque, in2 := 100.0, out => #data[54])
      { S7_Templates := "[SrcType := LReal, DestType := DInt]" } Convert(in := #data[54], out => "Unit1.EventsData".TelemetryContent[6].KVP[54].Value)
   END_RUNG
   // the same network as SCL:
   IF true AND false THEN "Unit1.EventsData".TelemetryContent[6].KVP[54].Value := 100; END_IF;
   IF true AND true THEN
       #data[54] := "Unit1.Em6.HmiInterface".cmMendrelCathodeFrontAxisZ.monitoring.actualTorque * 100.0;
       "Unit1.EventsData".TelemetryContent[6].KVP[54].Value := LREAL_TO_DINT(#data[54]);
   END_IF;
END_REGION

REGION Network 56: PDR Data55
   RUNG wire#powerrail
      Contact( true )
      wire#w1
      Contact( false )
      Move(in := 100, out1 => "Unit1.EventsData".TelemetryContent[6].KVP[55].Value)
   END_RUNG
   RUNG wire#w1
      Contact( true )
      { S7_Templates := "SrcType := LReal" } Mul(in1 := 0.0, in2 := 100.0, out => #data[55])
      { S7_Templates := "[SrcType := LReal, DestType := DInt]" } Convert(in := #data[55], out => "Unit1.EventsData".TelemetryContent[6].KVP[55].Value)
   END_RUNG
   // the same network as SCL:
   IF true AND false THEN "Unit1.EventsData".TelemetryContent[6].KVP[55].Value := 100; END_IF;
   IF true AND true THEN
       #data[55] := 0.0 * 100.0;
       "Unit1.EventsData".TelemetryContent[6].KVP[55].Value := LREAL_TO_DINT(#data[55]);
   END_IF;
END_REGION

REGION Network 57: PDR Data56 Stack Table Out Front AxisZ Actual Position
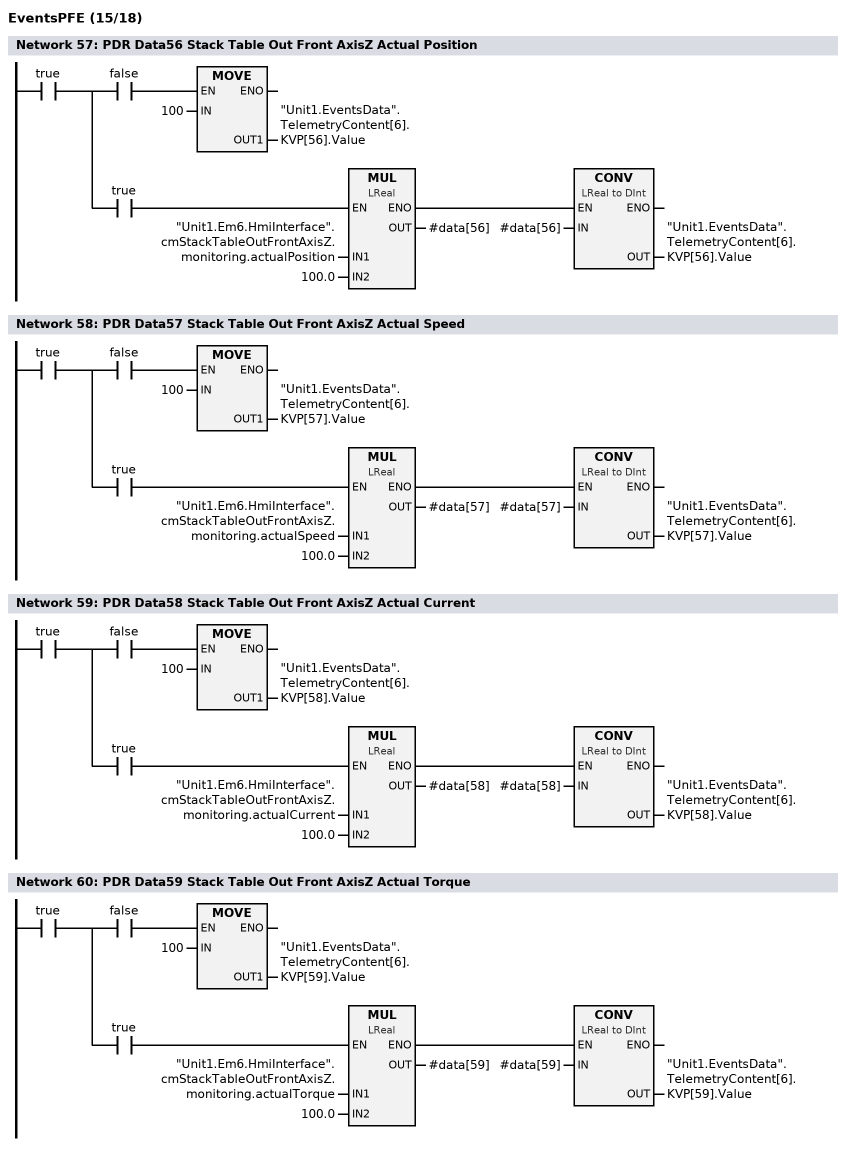
   RUNG wire#powerrail
      Contact( true )
      wire#w1
      Contact( false )
      Move(in := 100, out1 => "Unit1.EventsData".TelemetryContent[6].KVP[56].Value)
   END_RUNG
   RUNG wire#w1
      Contact( true )
      { S7_Templates := "SrcType := LReal" } Mul(in1 := "Unit1.Em6.HmiInterface".cmStackTableOutFrontAxisZ.monitoring.actualPosition, in2 := 100.0, out => #data[56])
      { S7_Templates := "[SrcType := LReal, DestType := DInt]" } Convert(in := #data[56], out => "Unit1.EventsData".TelemetryContent[6].KVP[56].Value)
   END_RUNG
   // the same network as SCL:
   IF true AND false THEN "Unit1.EventsData".TelemetryContent[6].KVP[56].Value := 100; END_IF;
   IF true AND true THEN
       #data[56] := "Unit1.Em6.HmiInterface".cmStackTableOutFrontAxisZ.monitoring.actualPosition * 100.0;
       "Unit1.EventsData".TelemetryContent[6].KVP[56].Value := LREAL_TO_DINT(#data[56]);
   END_IF;
END_REGION

REGION Network 58: PDR Data57 Stack Table Out Front AxisZ Actual Speed
   RUNG wire#powerrail
      Contact( true )
      wire#w1
      Contact( false )
      Move(in := 100, out1 => "Unit1.EventsData".TelemetryContent[6].KVP[57].Value)
   END_RUNG
   RUNG wire#w1
      Contact( true )
      { S7_Templates := "SrcType := LReal" } Mul(in1 := "Unit1.Em6.HmiInterface".cmStackTableOutFrontAxisZ.monitoring.actualSpeed, in2 := 100.0, out => #data[57])
      { S7_Templates := "[SrcType := LReal, DestType := DInt]" } Convert(in := #data[57], out => "Unit1.EventsData".TelemetryContent[6].KVP[57].Value)
   END_RUNG
   // the same network as SCL:
   IF true AND false THEN "Unit1.EventsData".TelemetryContent[6].KVP[57].Value := 100; END_IF;
   IF true AND true THEN
       #data[57] := "Unit1.Em6.HmiInterface".cmStackTableOutFrontAxisZ.monitoring.actualSpeed * 100.0;
       "Unit1.EventsData".TelemetryContent[6].KVP[57].Value := LREAL_TO_DINT(#data[57]);
   END_IF;
END_REGION

REGION Network 59: PDR Data58 Stack Table Out Front AxisZ Actual Current
   RUNG wire#powerrail
      Contact( true )
      wire#w1
      Contact( false )
      Move(in := 100, out1 => "Unit1.EventsData".TelemetryContent[6].KVP[58].Value)
   END_RUNG
   RUNG wire#w1
      Contact( true )
      { S7_Templates := "SrcType := LReal" } Mul(in1 := "Unit1.Em6.HmiInterface".cmStackTableOutFrontAxisZ.monitoring.actualCurrent, in2 := 100.0, out => #data[58])
      { S7_Templates := "[SrcType := LReal, DestType := DInt]" } Convert(in := #data[58], out => "Unit1.EventsData".TelemetryContent[6].KVP[58].Value)
   END_RUNG
   // the same network as SCL:
   IF true AND false THEN "Unit1.EventsData".TelemetryContent[6].KVP[58].Value := 100; END_IF;
   IF true AND true THEN
       #data[58] := "Unit1.Em6.HmiInterface".cmStackTableOutFrontAxisZ.monitoring.actualCurrent * 100.0;
       "Unit1.EventsData".TelemetryContent[6].KVP[58].Value := LREAL_TO_DINT(#data[58]);
   END_IF;
END_REGION

REGION Network 60: PDR Data59 Stack Table Out Front AxisZ Actual Torque
   RUNG wire#powerrail
      Contact( true )
      wire#w1
      Contact( false )
      Move(in := 100, out1 => "Unit1.EventsData".TelemetryContent[6].KVP[59].Value)
   END_RUNG
   RUNG wire#w1
      Contact( true )
      { S7_Templates := "SrcType := LReal" } Mul(in1 := "Unit1.Em6.HmiInterface".cmStackTableOutFrontAxisZ.monitoring.actualTorque, in2 := 100.0, out => #data[59])
      { S7_Templates := "[SrcType := LReal, DestType := DInt]" } Convert(in := #data[59], out => "Unit1.EventsData".TelemetryContent[6].KVP[59].Value)
   END_RUNG
   // the same network as SCL:
   IF true AND false THEN "Unit1.EventsData".TelemetryContent[6].KVP[59].Value := 100; END_IF;
   IF true AND true THEN
       #data[59] := "Unit1.Em6.HmiInterface".cmStackTableOutFrontAxisZ.monitoring.actualTorque * 100.0;
       "Unit1.EventsData".TelemetryContent[6].KVP[59].Value := LREAL_TO_DINT(#data[59]);
   END_IF;
END_REGION

REGION Network 61: PDR Data60
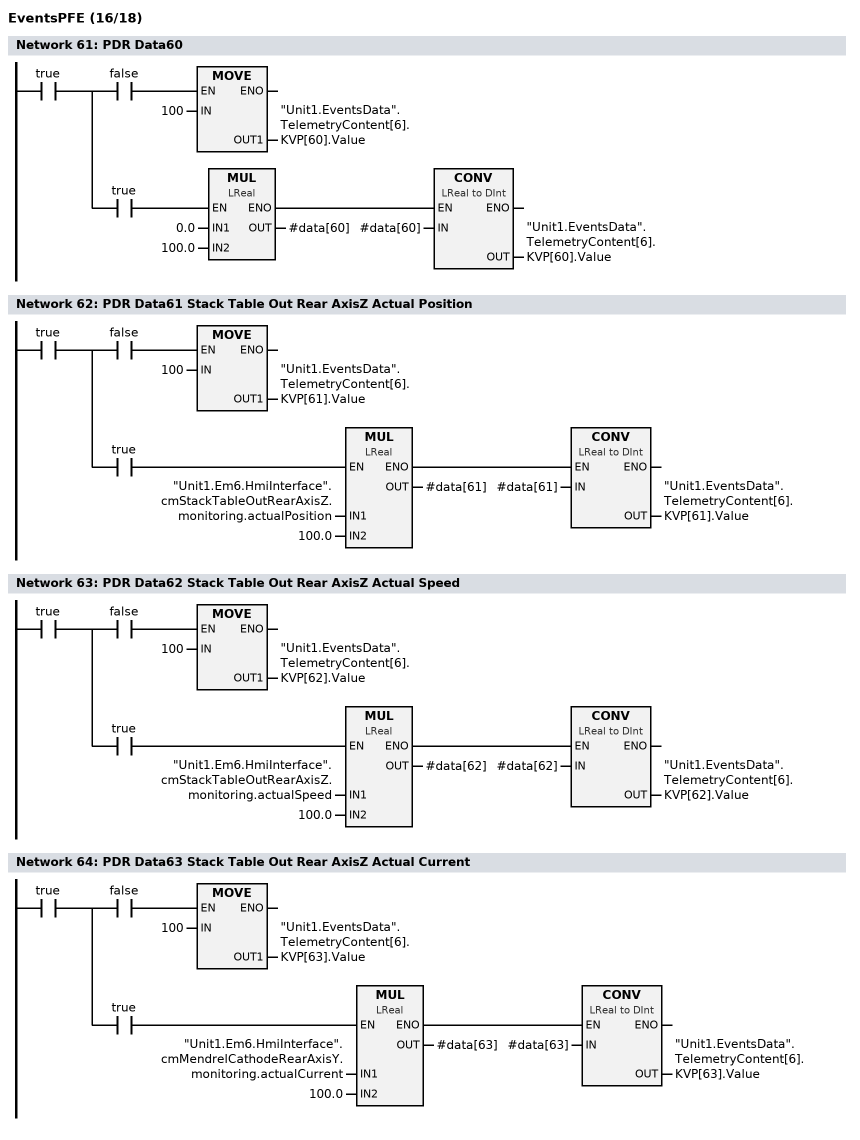
   RUNG wire#powerrail
      Contact( true )
      wire#w1
      Contact( false )
      Move(in := 100, out1 => "Unit1.EventsData".TelemetryContent[6].KVP[60].Value)
   END_RUNG
   RUNG wire#w1
      Contact( true )
      { S7_Templates := "SrcType := LReal" } Mul(in1 := 0.0, in2 := 100.0, out => #data[60])
      { S7_Templates := "[SrcType := LReal, DestType := DInt]" } Convert(in := #data[60], out => "Unit1.EventsData".TelemetryContent[6].KVP[60].Value)
   END_RUNG
   // the same network as SCL:
   IF true AND false THEN "Unit1.EventsData".TelemetryContent[6].KVP[60].Value := 100; END_IF;
   IF true AND true THEN
       #data[60] := 0.0 * 100.0;
       "Unit1.EventsData".TelemetryContent[6].KVP[60].Value := LREAL_TO_DINT(#data[60]);
   END_IF;
END_REGION

REGION Network 62: PDR Data61 Stack Table Out Rear AxisZ Actual Position
   RUNG wire#powerrail
      Contact( true )
      wire#w1
      Contact( false )
      Move(in := 100, out1 => "Unit1.EventsData".TelemetryContent[6].KVP[61].Value)
   END_RUNG
   RUNG wire#w1
      Contact( true )
      { S7_Templates := "SrcType := LReal" } Mul(in1 := "Unit1.Em6.HmiInterface".cmStackTableOutRearAxisZ.monitoring.actualPosition, in2 := 100.0, out => #data[61])
      { S7_Templates := "[SrcType := LReal, DestType := DInt]" } Convert(in := #data[61], out => "Unit1.EventsData".TelemetryContent[6].KVP[61].Value)
   END_RUNG
   // the same network as SCL:
   IF true AND false THEN "Unit1.EventsData".TelemetryContent[6].KVP[61].Value := 100; END_IF;
   IF true AND true THEN
       #data[61] := "Unit1.Em6.HmiInterface".cmStackTableOutRearAxisZ.monitoring.actualPosition * 100.0;
       "Unit1.EventsData".TelemetryContent[6].KVP[61].Value := LREAL_TO_DINT(#data[61]);
   END_IF;
END_REGION

REGION Network 63: PDR Data62 Stack Table Out Rear AxisZ Actual Speed
   RUNG wire#powerrail
      Contact( true )
      wire#w1
      Contact( false )
      Move(in := 100, out1 => "Unit1.EventsData".TelemetryContent[6].KVP[62].Value)
   END_RUNG
   RUNG wire#w1
      Contact( true )
      { S7_Templates := "SrcType := LReal" } Mul(in1 := "Unit1.Em6.HmiInterface".cmStackTableOutRearAxisZ.monitoring.actualSpeed, in2 := 100.0, out => #data[62])
      { S7_Templates := "[SrcType := LReal, DestType := DInt]" } Convert(in := #data[62], out => "Unit1.EventsData".TelemetryContent[6].KVP[62].Value)
   END_RUNG
   // the same network as SCL:
   IF true AND false THEN "Unit1.EventsData".TelemetryContent[6].KVP[62].Value := 100; END_IF;
   IF true AND true THEN
       #data[62] := "Unit1.Em6.HmiInterface".cmStackTableOutRearAxisZ.monitoring.actualSpeed * 100.0;
       "Unit1.EventsData".TelemetryContent[6].KVP[62].Value := LREAL_TO_DINT(#data[62]);
   END_IF;
END_REGION

REGION Network 64: PDR Data63 Stack Table Out Rear AxisZ Actual Current
   RUNG wire#powerrail
      Contact( true )
      wire#w1
      Contact( false )
      Move(in := 100, out1 => "Unit1.EventsData".TelemetryContent[6].KVP[63].Value)
   END_RUNG
   RUNG wire#w1
      Contact( true )
      { S7_Templates := "SrcType := LReal" } Mul(in1 := "Unit1.Em6.HmiInterface".cmMendrelCathodeRearAxisY.monitoring.actualCurrent, in2 := 100.0, out => #data[63])
      { S7_Templates := "[SrcType := LReal, DestType := DInt]" } Convert(in := #data[63], out => "Unit1.EventsData".TelemetryContent[6].KVP[63].Value)
   END_RUNG
   // the same network as SCL:
   IF true AND false THEN "Unit1.EventsData".TelemetryContent[6].KVP[63].Value := 100; END_IF;
   IF true AND true THEN
       #data[63] := "Unit1.Em6.HmiInterface".cmMendrelCathodeRearAxisY.monitoring.actualCurrent * 100.0;
       "Unit1.EventsData".TelemetryContent[6].KVP[63].Value := LREAL_TO_DINT(#data[63]);
   END_IF;
END_REGION

REGION Network 65: PDR Data64 Stack Table Out Rear AxisZ Actual Torque
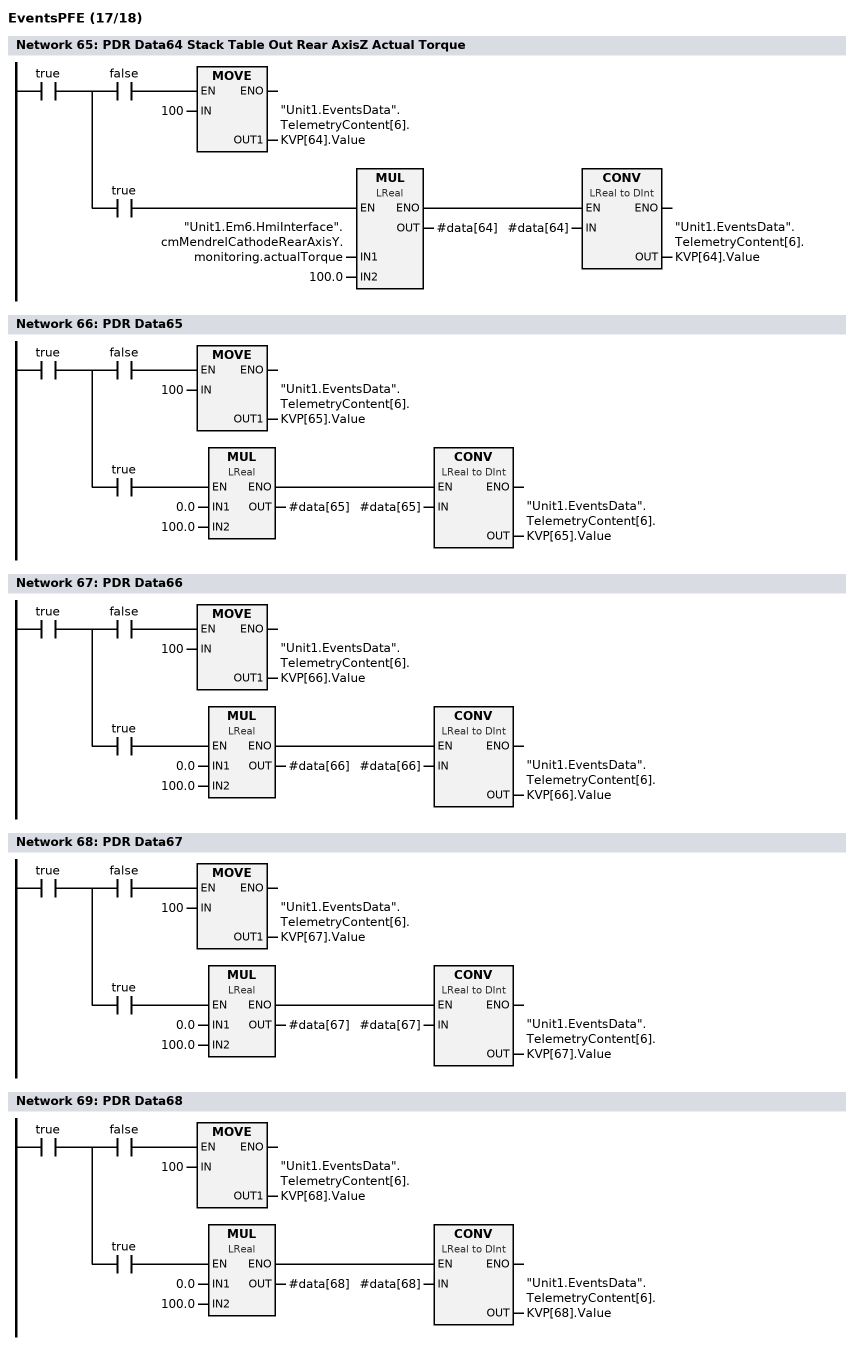
   RUNG wire#powerrail
      Contact( true )
      wire#w1
      Contact( false )
      Move(in := 100, out1 => "Unit1.EventsData".TelemetryContent[6].KVP[64].Value)
   END_RUNG
   RUNG wire#w1
      Contact( true )
      { S7_Templates := "SrcType := LReal" } Mul(in1 := "Unit1.Em6.HmiInterface".cmMendrelCathodeRearAxisY.monitoring.actualTorque, in2 := 100.0, out => #data[64])
      { S7_Templates := "[SrcType := LReal, DestType := DInt]" } Convert(in := #data[64], out => "Unit1.EventsData".TelemetryContent[6].KVP[64].Value)
   END_RUNG
   // the same network as SCL:
   IF true AND false THEN "Unit1.EventsData".TelemetryContent[6].KVP[64].Value := 100; END_IF;
   IF true AND true THEN
       #data[64] := "Unit1.Em6.HmiInterface".cmMendrelCathodeRearAxisY.monitoring.actualTorque * 100.0;
       "Unit1.EventsData".TelemetryContent[6].KVP[64].Value := LREAL_TO_DINT(#data[64]);
   END_IF;
END_REGION

REGION Network 66: PDR Data65
   RUNG wire#powerrail
      Contact( true )
      wire#w1
      Contact( false )
      Move(in := 100, out1 => "Unit1.EventsData".TelemetryContent[6].KVP[65].Value)
   END_RUNG
   RUNG wire#w1
      Contact( true )
      { S7_Templates := "SrcType := LReal" } Mul(in1 := 0.0, in2 := 100.0, out => #data[65])
      { S7_Templates := "[SrcType := LReal, DestType := DInt]" } Convert(in := #data[65], out => "Unit1.EventsData".TelemetryContent[6].KVP[65].Value)
   END_RUNG
   // the same network as SCL:
   IF true AND false THEN "Unit1.EventsData".TelemetryContent[6].KVP[65].Value := 100; END_IF;
   IF true AND true THEN
       #data[65] := 0.0 * 100.0;
       "Unit1.EventsData".TelemetryContent[6].KVP[65].Value := LREAL_TO_DINT(#data[65]);
   END_IF;
END_REGION

REGION Network 67: PDR Data66
   RUNG wire#powerrail
      Contact( true )
      wire#w1
      Contact( false )
      Move(in := 100, out1 => "Unit1.EventsData".TelemetryContent[6].KVP[66].Value)
   END_RUNG
   RUNG wire#w1
      Contact( true )
      { S7_Templates := "SrcType := LReal" } Mul(in1 := 0.0, in2 := 100.0, out => #data[66])
      { S7_Templates := "[SrcType := LReal, DestType := DInt]" } Convert(in := #data[66], out => "Unit1.EventsData".TelemetryContent[6].KVP[66].Value)
   END_RUNG
   // the same network as SCL:
   IF true AND false THEN "Unit1.EventsData".TelemetryContent[6].KVP[66].Value := 100; END_IF;
   IF true AND true THEN
       #data[66] := 0.0 * 100.0;
       "Unit1.EventsData".TelemetryContent[6].KVP[66].Value := LREAL_TO_DINT(#data[66]);
   END_IF;
END_REGION

REGION Network 68: PDR Data67
   RUNG wire#powerrail
      Contact( true )
      wire#w1
      Contact( false )
      Move(in := 100, out1 => "Unit1.EventsData".TelemetryContent[6].KVP[67].Value)
   END_RUNG
   RUNG wire#w1
      Contact( true )
      { S7_Templates := "SrcType := LReal" } Mul(in1 := 0.0, in2 := 100.0, out => #data[67])
      { S7_Templates := "[SrcType := LReal, DestType := DInt]" } Convert(in := #data[67], out => "Unit1.EventsData".TelemetryContent[6].KVP[67].Value)
   END_RUNG
   // the same network as SCL:
   IF true AND false THEN "Unit1.EventsData".TelemetryContent[6].KVP[67].Value := 100; END_IF;
   IF true AND true THEN
       #data[67] := 0.0 * 100.0;
       "Unit1.EventsData".TelemetryContent[6].KVP[67].Value := LREAL_TO_DINT(#data[67]);
   END_IF;
END_REGION

REGION Network 69: PDR Data68
   RUNG wire#powerrail
      Contact( true )
      wire#w1
      Contact( false )
      Move(in := 100, out1 => "Unit1.EventsData".TelemetryContent[6].KVP[68].Value)
   END_RUNG
   RUNG wire#w1
      Contact( true )
      { S7_Templates := "SrcType := LReal" } Mul(in1 := 0.0, in2 := 100.0, out => #data[68])
      { S7_Templates := "[SrcType := LReal, DestType := DInt]" } Convert(in := #data[68], out => "Unit1.EventsData".TelemetryContent[6].KVP[68].Value)
   END_RUNG
   // the same network as SCL:
   IF true AND false THEN "Unit1.EventsData".TelemetryContent[6].KVP[68].Value := 100; END_IF;
   IF true AND true THEN
       #data[68] := 0.0 * 100.0;
       "Unit1.EventsData".TelemetryContent[6].KVP[68].Value := LREAL_TO_DINT(#data[68]);
   END_IF;
END_REGION

REGION Network 70: PDR Data69
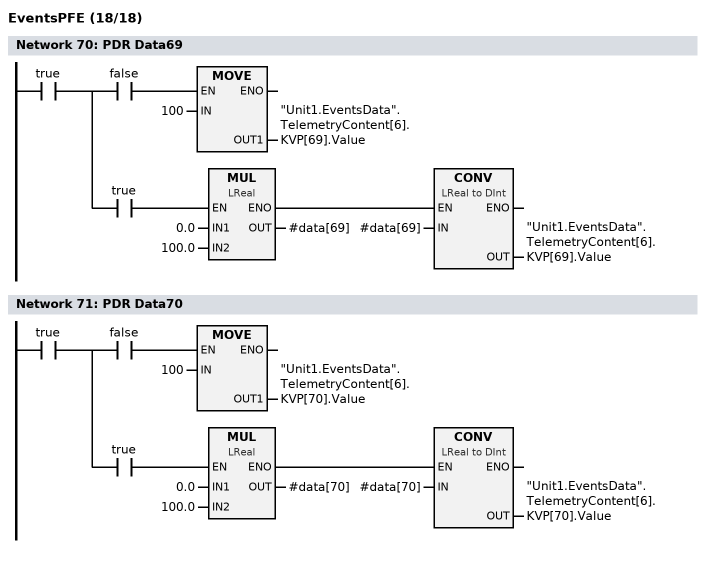
   RUNG wire#powerrail
      Contact( true )
      wire#w1
      Contact( false )
      Move(in := 100, out1 => "Unit1.EventsData".TelemetryContent[6].KVP[69].Value)
   END_RUNG
   RUNG wire#w1
      Contact( true )
      { S7_Templates := "SrcType := LReal" } Mul(in1 := 0.0, in2 := 100.0, out => #data[69])
      { S7_Templates := "[SrcType := LReal, DestType := DInt]" } Convert(in := #data[69], out => "Unit1.EventsData".TelemetryContent[6].KVP[69].Value)
   END_RUNG
   // the same network as SCL:
   IF true AND false THEN "Unit1.EventsData".TelemetryContent[6].KVP[69].Value := 100; END_IF;
   IF true AND true THEN
       #data[69] := 0.0 * 100.0;
       "Unit1.EventsData".TelemetryContent[6].KVP[69].Value := LREAL_TO_DINT(#data[69]);
   END_IF;
END_REGION

REGION Network 71: PDR Data70
   RUNG wire#powerrail
      Contact( true )
      wire#w1
      Contact( false )
      Move(in := 100, out1 => "Unit1.EventsData".TelemetryContent[6].KVP[70].Value)
   END_RUNG
   RUNG wire#w1
      Contact( true )
      { S7_Templates := "SrcType := LReal" } Mul(in1 := 0.0, in2 := 100.0, out => #data[70])
      { S7_Templates := "[SrcType := LReal, DestType := DInt]" } Convert(in := #data[70], out => "Unit1.EventsData".TelemetryContent[6].KVP[70].Value)
   END_RUNG
   // the same network as SCL:
   IF true AND false THEN "Unit1.EventsData".TelemetryContent[6].KVP[70].Value := 100; END_IF;
   IF true AND true THEN
       #data[70] := 0.0 * 100.0;
       "Unit1.EventsData".TelemetryContent[6].KVP[70].Value := LREAL_TO_DINT(#data[70]);
   END_IF;
END_REGION
END_FUNCTION_BLOCK
